ABB RAPID module: PRG_MVT.mod

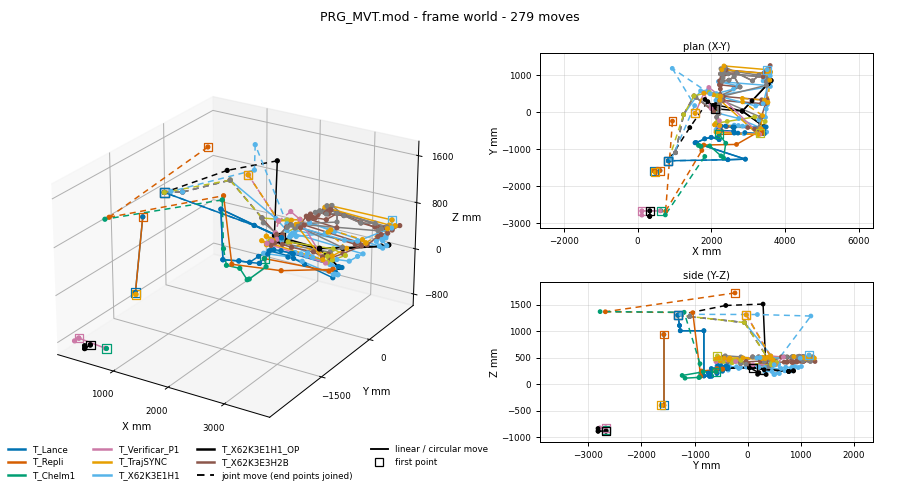
[picture p0: tool path of PRG_MVT.mod in frame world, 279 of 334 moves have a stored position in this frame; points joined in program order, loops and branches not executed]
%%%
  VERSION:1
  LANGUAGE:ENGLISH
%%%

MODULE PRG_MVT
  !********************************************
  !*                                          *
  !*      ABB--PROMIA--50.xx                  *
  !*                                          *
  !* Module Programme de mouvement            *
  !* Baie de commande de type IRC5            *
  !* Mono-robot                               *
  !********************************************
  !
  !=========================
  ! Donnees de type tooldata
  !=========================
  ! Outil par défaut pour T_Repli, T_Lance et trajs de Maintenance
  ! Les données de charge sont à renseigner !
  TASK PERS tooldata Tool_defaut:=[TRUE,[[0,0,0],[1,0,0,0]],[274,[0,0,0.001],[1,0,0,0],24.55,73.06,97.5]];
  ! Les données de charge et référentiels sont à renseigner !
  TASK PERS tooldata Tool_Pince1:=[TRUE,[[-1102.56,2.69854,432.58],[0.000350004,0,1,0]],[274,[0,0,0.001],[1,0,0,0],24.55,73.06,97.5]];
  TASK PERS tooldata Tool_Pince2:=[TRUE,[[0,0,0],[1,0,0,0]],[0.001,[0,0,0.001],[1,0,0,0],0,0,0]];
  TASK PERS tooldata Tool_Pince3:=[TRUE,[[0,0,0],[1,0,0,0]],[0.001,[0,0,0.001],[1,0,0,0],0,0,0]];
  TASK PERS tooldata Tool_Pince4:=[TRUE,[[0,0,0],[1,0,0,0]],[0.001,[0,0,0.001],[1,0,0,0],0,0,0]];
	TASK PERS tooldata Tool_etalonR1:=[TRUE,[[0,0,0],[1,0,0,0]],[0.001,[0,0,0.001],[1,0,0,0],0,0,0]];
  TASK PERS tooldata Tool_R1:=[TRUE,[[0,0,0],[1,0,0,0]],[0.001,[0,0,0.001],[1,0,0,0],0,0,0]];
  TASK PERS tooldata tMaxMotion:=[TRUE,[[-1102.56,2.69854,432.58],[0.000350004,0,1,0]],[0.001,[0,0,0.001],[1,0,0,0],0,0,0]];
  TASK PERS tooldata toolAtual:=[TRUE,[[0,0,0],[1,0,0,0]],[274,[0,0,0.001],[1,0,0,0],24.55,73.06,97.5]];
  PERS tooldata Temp_tool:=[TRUE,[[0,0,0],[1,0,0,0]],[0.001,[0,0,0.001],[1,0,0,0],0,0,0]];
  TASK PERS tooldata Pince1:=[TRUE,[[-1100.74,0,428.94],[0,0,1,0]],[274,[0,0,0.001],[1,0,0,0],24.55,73.06,97.5]];
  !
  !=========================
  ! Donnees de type wobjdata
  !=========================
  PERS wobjdata wobj_X62:=[FALSE,TRUE,"",[[0,0,0],[1,0,0,0]],[[2652.5,-1847.7,-1638.89],[0.737289,0.000738386,0.00238165,0.675573]]];
  TASK PERS wobjdata w_A11:=[FALSE,TRUE,"",[[723.52,3.59082,586.622],[0.104509,0.031933,0.994006,-0.00335437]],[[0,0,0],[0,1,0,0]]];
  TASK PERS wobjdata W_A21:=[FALSE,TRUE,"",[[723.52,3.59,586.62],[1,0,0,0]],[[0,0,0],[0,1,0,0]]];
  PERS wobjdata Temp_wobj:=[FALSE,TRUE,"",[[0,0,0],[1,0,0,0]],[[0,0,0],[1,0,0,0]]];
  PERS wobjdata Temp2_wobj:=[FALSE,TRUE,"",[[0,0,0],[1,0,0,0]],[[0,0,0],[1,0,0,0]]];
  TASK PERS wobjdata wobjAtual:=[FALSE,TRUE,"",[[0,0,0],[1,0,0,0]],[[0,0,0],[1,0,0,0]]];
  PERS wobjdata wobj_XDF:=[False,True,"",[[2664.9690,-1849.2940,-1633.2210],[0.737546,-0.004241,-0.002957,0.675277]],[[0,0,0],[1,0,0,0]]];
  !
  !=========================
  ! Donnees de type robtarget
  !=========================
  CONST robtarget pInicioX62_Pinca1:=[[366.51,1868.19,2935],[0.00946049,0.00387218,0.00595509,0.99993],[-1,-1,0,0],[29.4996,9E+09,9E+09,9E+09,9E+09,9E+09]];
  CONST robtarget pReferenciaPinca1:=[[117.16,-2786.22,-820.12],[0.578822,-0.00575624,0.000186763,-0.815434],[-1,-1,0,0],[72.8969,9E+09,9E+09,9E+09,9E+09,9E+09]];
  CONST robtarget pFresaPinca1:=[[330.76,-2818.92,-832.36],[0.67068,-0.00156521,-0.011854,-0.741651],[-1,0,0,0],[22.3121,9E+09,9E+09,9E+09,9E+09,9E+09]];
  CONST robtarget pTrocaEletrodosPinca1:=[[634.22,-2665.42,-865.34],[0.767575,-0.0054113,0.00150274,-0.640935],[-1,-1,0,0],[129.398,9E+09,9E+09,9E+09,9E+09,9E+09]];
  !

  !
  !=========================
  ! Donnees de type robtarget
  !=========================
  !Option Securité
  CONST jointtarget pPSync:=[[-74.4391,71.8518,8.78224,-3.78008,9.21547,38.5548],[72.8966,9E+09,9E+09,9E+09,9E+09,9E+09]];
  !
  !=========================
  ! Donnees de type bool
  !=========================
  PERS bool EPSRequest:=FALSE;
  !
  !-----------------------
  !     T_X62K3E1H1
  !-----------------------
  CONST robtarget lscs1002841400:=[[1321.80,-611.52,1989.42],[0.57763,-0.0127115,0.00458018,-0.816187],[-1,-1,0,0],[34.9983,9E+09,9E+09,9E+09,9E+09,9E+09]];
  CONST robtarget lscs1002841500:=[[1421.03,-636.06,1985.03],[0.577855,-0.0132046,0.00335794,-0.816026],[-1,-1,0,0],[34.9978,9E+09,9E+09,9E+09,9E+09,9E+09]];
  CONST robtarget lscs1002841900:=[[2124.39,-642.18,1983.84],[0.696596,0.0227135,0.0233793,-0.716723],[0,0,0,0],[34.9999,9E+09,9E+09,9E+09,9E+09,9E+09]];
  CONST robtarget lscs1002842000:=[[2228.68,-635.15,1986.45],[0.695583,0.0213858,0.0221666,-0.717786],[0,0,0,0],[35.0049,9E+09,9E+09,9E+09,9E+09,9E+09]];
  CONST robtarget lscs1002842300:=[[2641.55,-631.88,1984.23],[0.78191,0.0244769,0.0194947,-0.622606],[0,0,0,0],[20,9E+09,9E+09,9E+09,9E+09,9E+09]];
  CONST robtarget lscs1002842400:=[[2740.12,-630.61,1983.50],[0.787083,0.0248153,0.0202104,-0.616017],[0,0,0,0],[34.9988,9E+09,9E+09,9E+09,9E+09,9E+09]];
  CONST robtarget lscs1003265500:=[[1660.38,-715.96,1974.39],[0.623818,6.28508E-06,9.80078E-06,-0.781569],[0,-1,0,0],[35,9E+09,9E+09,9E+09,9E+09,9E+09]];
  CONST robtarget lscs1003265600:=[[1771.68,-715.35,1974.08],[0.641583,2.04864E-06,1.74234E-06,-0.767054],[0,-1,0,0],[35,9E+09,9E+09,9E+09,9E+09,9E+09]];
  CONST robtarget lscs1003265800:=[[2000.05,-716.75,1973.15],[0.67611,2.28831E-06,2.51046E-06,-0.736801],[0,-1,0,0],[34.9998,9E+09,9E+09,9E+09,9E+09,9E+09]];
  CONST robtarget lscs1003265900:=[[2103.17,-716.71,1973.07],[0.692842,6.80056E-06,1.10347E-05,-0.72109],[0,-1,0,0],[34.9998,9E+09,9E+09,9E+09,9E+09,9E+09]];
  CONST robtarget lscs1003266000:=[[2247.94,-712.34,1973.89],[0.709194,1.03549E-05,1.67342E-05,-0.705013],[0,-1,0,0],[34.9997,9E+09,9E+09,9E+09,9E+09,9E+09]];
  CONST robtarget lscs1003266100:=[[2332.06,-711.17,1972.75],[0.725199,1.11717E-05,1.69368E-05,-0.688539],[0,-1,0,0],[35,9E+09,9E+09,9E+09,9E+09,9E+09]];
  CONST robtarget lscs1003266200:=[[2415.91,-712.40,1971.62],[0.740802,6.31206E-07,-8.02992E-07,-0.671724],[0,-1,0,0],[35.0003,9E+09,9E+09,9E+09,9E+09,9E+09]];
  CONST robtarget lscs1003267400:=[[2515.38,-713.65,1970.65],[0.75603,-5.40779E-06,-9.51741E-06,-0.654537],[0,-1,0,0],[35,9E+09,9E+09,9E+09,9E+09,9E+09]];
  CONST robtarget lscs1003267500:=[[2614.89,-713.96,1971.44],[0.770849,8.75642E-06,1.09504E-05,-0.637018],[0,-1,0,0],[34.9997,9E+09,9E+09,9E+09,9E+09,9E+09]];
  CONST robtarget lscs1003267600:=[[2753.83,-713.47,1973.81],[0.787351,1.19686E-07,-7.7226E-06,-0.616505],[0,-1,0,0],[34.9996,9E+09,9E+09,9E+09,9E+09,9E+09]];
  CONST robtarget lscs1003267700:=[[2860.11,-710.59,1972.43],[0.787349,7.34808E-06,1.07537E-05,-0.616508],[0,-1,0,0],[35.0003,9E+09,9E+09,9E+09,9E+09,9E+09]];
  CONST robtarget lscs1003268200:=[[2954.09,-709.12,1972.24],[0.797982,-2.34679E-06,-6.61137E-06,-0.602681],[0,-1,0,0],[34.9997,9E+09,9E+09,9E+09,9E+09,9E+09]];
  CONST robtarget lscs1004621400:=[[1320.78,-635.11,1988.81],[0.577563,-0.00428276,0.010528,-0.816267],[-1,-1,0,0],[34.9983,9E+09,9E+09,9E+09,9E+09,9E+09]];
  CONST robtarget lscs1005331700:=[[1371.89,-717.33,1972.12],[0.595248,1.0937E-05,1.49243E-05,-0.803542],[-1,-1,0,0],[35.0037,9E+09,9E+09,9E+09,9E+09,9E+09]];
  CONST robtarget lscs2002842100:=[[2131.94,651.05,1966.73],[0.600981,-0.019579,-0.0260102,-0.7986],[0,-1,0,0],[25.7552,9E+09,9E+09,9E+09,9E+09,9E+09]];
  CONST robtarget lscs2002842200:=[[2234.34,649.61,1967.17],[0.613888,-0.0189544,-0.024229,-0.788794],[0,-1,0,0],[35.0005,9E+09,9E+09,9E+09,9E+09,9E+09]];
  CONST robtarget lscs2002842500:=[[2637.04,646.84,1973.10],[0.920442,-0.0269256,-0.00783123,-0.389872],[0,-1,-1,0],[33.1616,9E+09,9E+09,9E+09,9E+09,9E+09]];
  CONST robtarget lscs2003266400:=[[1657.98,727.29,1955.98],[0.356059,6.94468E-07,9.41827E-06,-0.934464],[0,0,0,0],[34.9945,9E+09,9E+09,9E+09,9E+09,9E+09]];
  CONST robtarget lscs2003266500:=[[1770.24,729.39,1956.83],[0.388522,1.29051E-06,-2.04438E-06,-0.92144],[0,0,0,0],[34.9997,9E+09,9E+09,9E+09,9E+09,9E+09]];
  CONST robtarget lscs2003266700:=[[1997.48,731.61,1956.90],[0.4602,4.00795E-06,-1.13671E-05,-0.887816],[0,0,0,0],[35.0891,9E+09,9E+09,9E+09,9E+09,9E+09]];
  CONST robtarget lscs2003266800:=[[2112.90,726.36,1955.43],[0.601155,1.22632E-06,9.81834E-06,-0.799133],[0,0,0,0],[35.0002,9E+09,9E+09,9E+09,9E+09,9E+09]];
  CONST robtarget lscs2003266900:=[[2249.72,730.07,1955.35],[0.614381,1.7781E-06,2.41043E-05,-0.789009],[0,0,0,0],[34.9999,9E+09,9E+09,9E+09,9E+09,9E+09]];
  CONST robtarget lscs2003267000:=[[2334.19,729.87,1957.44],[0.614386,-1.46543E-06,1.51219E-06,-0.789006],[0,0,0,0],[35.002,9E+09,9E+09,9E+09,9E+09,9E+09]];
  CONST robtarget lscs2003267100:=[[2418.69,727.31,1957.28],[0.670217,2.34267E-06,1.10938E-05,-0.742166],[0,0,0,0],[35,9E+09,9E+09,9E+09,9E+09,9E+09]];
  CONST robtarget lscs2003267800:=[[2517.33,728.02,1957.52],[0.712352,3.39692E-06,1.72802E-05,-0.701822],[0,0,0,0],[35,9E+09,9E+09,9E+09,9E+09,9E+09]];
  CONST robtarget lscs2003267900:=[[2618.90,732.56,1958.73],[0.92597,1.3493E-05,8.03361E-06,-0.377598],[0,-1,-1,0],[50.0003,9E+09,9E+09,9E+09,9E+09,9E+09]];
  CONST robtarget lscsd004573702:=[[1500.55,728.22,1952.50],[0.327808,2.82413E-06,-3.88473E-07,-0.944744],[0,0,0,0],[35.0009,9E+09,9E+09,9E+09,9E+09,9E+09]];
  CONST robtarget lscsg004573701:=[[1490.46,-715.35,1972.01],[0.605617,0.0139801,0.0105122,-0.795564],[-1,0,0,0],[34.9991,9E+09,9E+09,9E+09,9E+09,9E+09]];
  CONST robtarget lspac002878500:=[[1419.00,-536.94,1995.23],[0.572412,-0.0117175,0.00271518,-0.819878],[0,-1,0,0],[24.6351,9E+09,9E+09,9E+09,9E+09,9E+09]];
  CONST robtarget lspac002878600:=[[1417.58,-399.17,2001.89],[0.554961,-0.011186,0.00127143,-0.8318],[0,-1,0,0],[27.0922,9E+09,9E+09,9E+09,9E+09,9E+09]];
  CONST robtarget lspac002878700:=[[1416.53,-283.20,2005.54],[0.539023,-0.00172498,0.00603882,-0.842268],[0,-1,0,0],[22.9219,9E+09,9E+09,9E+09,9E+09,9E+09]];
  CONST robtarget lspac002878800:=[[1416.52,-204.20,2006.05],[0.527512,-0.00580073,0.00167739,-0.849526],[0,-1,0,0],[20.8186,9E+09,9E+09,9E+09,9E+09,9E+09]];

  CONST robtarget lspac002878900:=[[1416.87,-59.54,2005.71],[0.445099,0.000472,0.001718,-0.89548],[0,0,0,0],[35.002,9E+09,9E+09,9E+09,9E+09,9E+09]];
  CONST robtarget lspac002879000:=[[1416.21,53.99,2003.54],[0.445095,-0.001082,-0.001403,-0.895482],[0,-1,0,0],[27.999,9E+09,9E+09,9E+09,9E+09,9E+09]];
  CONST robtarget lspac002879100:=[[1417.29,167.25,2000.96],[0.418464,-0.003529,-0.007686,-0.908194],[0,-1,0,0],[35,9E+09,9E+09,9E+09,9E+09,9E+09]];
  CONST robtarget lspac002879200:=[[1416.66,280.75,1998.11],[0.370926,-0.005338,-0.013272,-0.928552],[0,-1,0,0],[35,9E+09,9E+09,9E+09,9E+09,9E+09]];
  CONST robtarget lspac002879300:=[[1416.64,393.28,1993.21],[0.370888,-0.007028,-0.017515,-0.928486],[0,-1,0,0],[35.004,9E+09,9E+09,9E+09,9E+09,9E+09]];
  CONST robtarget lspac002879400:=[[1417.48,505.46,1988.3],[0.371815,-0.009151,-0.022849,-0.927981],[0,-1,0,0],[35.002,9E+09,9E+09,9E+09,9E+09,9E+09]];
  CONST robtarget lscs2002841700:=[[1425.2,650.88,1974.99],[0.292836,-0.009125,-0.029745,-0.955656],[0,-1,0,0],[35,9E+09,9E+09,9E+09,9E+09,9E+09]];
  CONST robtarget lscs2004621500:=[[1322.81,651.07,1978.03],[0.285706,-0.009516,-0.031739,-0.957744],[0,-1,0,0],[37.176,9E+09,9E+09,9E+09,9E+09,9E+09]];
  CONST robtarget lscs2002841600:=[[1322.39,627.55,1981.36],[0.302378,-0.010051,-0.031649,-0.95261],[0,-1,0,0],[35,9E+09,9E+09,9E+09,9E+09,9E+09]];
  CONST robtarget lspac002883300:=[[1326.62,507.5,1989.98],[0.308491,-0.007592,-0.023435,-0.950908],[0,-1,0,0],[23.854,9E+09,9E+09,9E+09,9E+09,9E+09]];
  CONST robtarget lspac002883200:=[[1325.86,394.19,1995.58],[0.331525,-0.006266,-0.017813,-0.943257],[0,-1,0,0],[23.958,9E+09,9E+09,9E+09,9E+09,9E+09]];

  CONST robtarget lspac002883100:=[[1325.42,281.32,1997.89],[0.419379,-0.005519,-0.011953,-0.907716],[0,-1,0,0],[25.495,25.495,9E+09,9E+09,9E+09,9E+09]];
  CONST robtarget lspac002882400:=[[1321.76,-509.09,1996.03],[0.531284,-0.00843427,0.00739349,-0.84712],[0,-1,0,0],[35.0007,9E+09,9E+09,9E+09,9E+09,9E+09]];
  CONST robtarget lspac002882500:=[[1324.54,-396.08,2000.52],[0.51375,-0.00327198,-0.0104843,-0.85787],[0,0,0,0],[34.9986,9E+09,9E+09,9E+09,9E+09,9E+09]];
  CONST robtarget lspac002882600:=[[1324.67,-284.50,2002.23],[0.496324,0.000459301,-0.00172718,-0.868135],[0,0,0,0],[34.9989,9E+09,9E+09,9E+09,9E+09,9E+09]];
  CONST robtarget lspac002882700:=[[1324.62,-171.83,2005.66],[0.478463,-0.00395536,-0.0119621,-0.878018],[0,-1,0,0],[24.4112,9E+09,9E+09,9E+09,9E+09,9E+09]];
  CONST robtarget lspac002882800:=[[1324.87,-57.50,2005.46],[0.460554,-0.0108643,-0.00417129,-0.887556],[0,-1,0,0],[35.0038,9E+09,9E+09,9E+09,9E+09,9E+09]];
  CONST robtarget lspac002882900:=[[1324.13,55.63,2003.75],[0.44275,-0.00105814,-0.00139436,-0.896644],[0,-1,0,0],[20.988,9E+09,9E+09,9E+09,9E+09,9E+09]];
  CONST robtarget lspac002883000:=[[1324.03,167.68,2002.17],[0.419385,-0.00274683,-0.00713244,-0.907777],[0,-1,0,0],[19.1411,9E+09,9E+09,9E+09,9E+09,9E+09]];
  CONST robtarget lspac002900900:=[[2226.97,-511.07,1992.43],[0.695722,0.0173592,0.0179165,-0.717878],[0,0,0,0],[35.0017,9E+09,9E+09,9E+09,9E+09,9E+09]];
  CONST robtarget lspac002901000:=[[2226.48,-365.82,1995.55],[0.696043,0.0128999,0.0133004,-0.717761],[0,0,0,0],[34.9992,9E+09,9E+09,9E+09,9E+09,9E+09]];
  CONST robtarget lspac002901100:=[[2225.60,-228.43,1999.39],[0.69581,0.00731454,0.00755639,-0.718149],[0,0,0,0],[35.0004,9E+09,9E+09,9E+09,9E+09,9E+09]];
  CONST robtarget lspac002901300:=[[2225.20,24.47,1997.06],[0.695924,-0.00113677,-0.00115838,-0.718113],[0,-1,0,0],[35.0004,9E+09,9E+09,9E+09,9E+09,9E+09]];
  CONST robtarget lspac002901600:=[[2225.18,226.53,1992.98],[0.695884,-0.00731719,-0.00753954,-0.718077],[0,-1,0,0],[35.0003,9E+09,9E+09,9E+09,9E+09,9E+09]];
  CONST robtarget lspac002901700:=[[2227.57,364.45,1984.47],[0.695822,-0.0128824,-0.0132698,-0.717977],[0,-1,0,0],[35.0013,9E+09,9E+09,9E+09,9E+09,9E+09]];
  CONST robtarget lspac002901800:=[[2227.15,509.55,1976.50],[0.614039,-0.0153147,-0.0196554,-0.788882],[0,-1,0,0],[34.9978,9E+09,9E+09,9E+09,9E+09,9E+09]];
  CONST robtarget lspac002904100:=[[2126.95,-510.92,1993.00],[0.702146,-0.00802476,-0.0133731,-0.711862],[0,-1,0,0],[34.998,9E+09,9E+09,9E+09,9E+09,9E+09]];
  CONST robtarget lspac002904200:=[[2129.65,-364.85,2000.21],[0.7056,-0.00721348,-0.00638237,-0.708545],[0,-1,0,0],[34.9979,9E+09,9E+09,9E+09,9E+09,9E+09]];
  CONST robtarget lspac002904300:=[[2129.80,-227.65,1999.07],[0.714409,0.00750987,0.00734911,-0.69965],[0,0,0,0],[22.0001,9E+09,9E+09,9E+09,9E+09,9E+09]];
  CONST robtarget lspac002904400:=[[2132.73,-25.26,1998.55],[0.682213,0.00111235,0.00119395,-0.731152],[0,0,0,0],[20.0001,9E+09,9E+09,9E+09,9E+09,9E+09]];
  CONST robtarget lspac002904600:=[[2133.65,228.53,1991.11],[0.682136,-0.00715952,-0.00768831,-0.73115],[0,-1,0,0],[23.0024,9E+09,9E+09,9E+09,9E+09,9E+09]];
  CONST robtarget lspac002904700:=[[2132.48,364.88,1986.15],[0.682017,-0.0126149,-0.0135198,-0.731103],[0,-1,0,0],[21.9995,9E+09,9E+09,9E+09,9E+09,9E+09]];
  CONST robtarget lspac002904800:=[[2133.45,510.43,1978.85],[0.681915,-0.0169944,-0.0182283,-0.731007],[0,-1,0,0],[20.5101,9E+09,9E+09,9E+09,9E+09,9E+09]];
  CONST robtarget lspac002905100:=[[2739.39,-510.19,1990.50],[0.787183,0.0196481,0.015397,-0.616215],[0,0,0,0],[34.9996,9E+09,9E+09,9E+09,9E+09,9E+09]];
  CONST robtarget lspac002906100:=[[2644.16,-510.46,1992.58],[0.793004,0.0197938,0.0151959,-0.608706],[0,0,0,0],[19.9993,9E+09,9E+09,9E+09,9E+09,9E+09]];
  CONST robtarget lspac002906200:=[[2643.42,-365.01,1995.40],[0.80405,0.0149065,0.0110176,-0.594273],[0,0,0,0],[30.3308,9E+09,9E+09,9E+09,9E+09,9E+09]];
  CONST robtarget lspac002906300:=[[2642.81,-227.08,2000.09],[0.814671,0.00856781,0.00608173,-0.579829],[0,0,-1,0],[38.4896,9E+09,9E+09,9E+09,9E+09,9E+09]];
  CONST robtarget lspac002906400:=[[2639.69,-24.86,1997.79],[0.835042,0.00138016,0.000921054,-0.550184],[0,-1,-1,0],[31.1701,9E+09,9E+09,9E+09,9E+09,9E+09]];
  CONST robtarget lspac002906600:=[[2642.07,228.52,1996.03],[0.854261,-0.00895447,-0.00544438,-0.51974],[0,-1,-1,0],[56.311,9E+09,9E+09,9E+09,9E+09,9E+09]];
  CONST robtarget lspac002906700:=[[2642.16,368.74,1991.45],[0.877971,-0.0162117,-0.00882183,-0.478359],[0,-1,-1,0],[25.0003,9E+09,9E+09,9E+09,9E+09,9E+09]];
  CONST robtarget lspac002906800:=[[2640.35,507.33,1982.42],[0.904527,-0.0225527,-0.010627,-0.425687],[0,-1,-1,0],[29.1146,9E+09,9E+09,9E+09,9E+09,9E+09]];
  CONST robtarget lspac006169900:=[[2225.43,89.14,1997.34],[0.695931,-0.00294883,-0.00302088,-0.718096],[0,-1,0,0],[35.0021,9E+09,9E+09,9E+09,9E+09,9E+09]];
  CONST robtarget lspac006170200:=[[2133.71,90.17,1997.24],[0.6822,-0.00290099,-0.00312195,-0.731154],[0,-1,0,0],[21.9945,9E+09,9E+09,9E+09,9E+09,9E+09]];
  CONST robtarget lspac006170400:=[[2641.02,91.45,1996.56],[0.844807,-0.0035688,-0.00227158,-0.535055],[0,-1,-1,0],[31.1277,9E+09,9E+09,9E+09,9E+09,9E+09]];
  CONST robtarget lspac006170500:=[[2226.35,-90.87,1999.36],[0.695897,0.00294943,0.00305218,-0.718129],[0,0,0,0],[34.9995,9E+09,9E+09,9E+09,9E+09,9E+09]];
  CONST robtarget lspac006170800:=[[2134.22,-89.69,2000.26],[0.720063,0.00306425,0.00294629,-0.693896],[0,0,0,0],[22,9E+09,9E+09,9E+09,9E+09,9E+09]];
  CONST robtarget lspac006171000:=[[2641.20,-82.11,1999.25],[0.824987,0.00352259,0.00243168,-0.565135],[0,0,-1,0],[38.713,9E+09,9E+09,9E+09,9E+09,9E+09]];
  !-----------------------
  !    T_X62K3E1H1_OP
  !-----------------------
  CONST robtarget lscs1003265700:=[[1886.36,-714.00,1973.66],[0.653882,-1.55351E-06,-1.78434E-06,-0.756597],[0,-1,0,0],[75.0001,9E+09,9E+09,9E+09,9E+09,9E+09]];
  CONST robtarget lscs2003266600:=[[1884.13,727.83,1956.34],[0.460207,5.49601E-07,1.78346E-06,-0.887812],[0,0,0,0],[74.9997,9E+09,9E+09,9E+09,9E+09,9E+09]];
  !-----------------------
  !    T_X62K3E23H2
  !-----------------------
  CONST robtarget lscs1002838100:=[[1326.03,-548.67,2179.62],[0.529877,0.0162447,0.0240929,-0.847577],[-1,0,0,0],[35.0008,9E+09,9E+09,9E+09,9E+09,9E+09]];
  CONST robtarget lscs1002838200:=[[1420.36,-572.64,2182.13],[0.520361,0.0154283,0.0248866,-0.853444],[0,0,0,0],[35.0001,9E+09,9E+09,9E+09,9E+09,9E+09]];
  CONST robtarget lscs1002838900:=[[2127.03,-573.84,2183.93],[0.703375,0.0176685,0.0238462,-0.710199],[0,0,0,0],[34.9991,9E+09,9E+09,9E+09,9E+09,9E+09]];
  CONST robtarget lscs1002839000:=[[2230.97,-578.10,2182.31],[0.695615,0.0204629,0.021045,-0.717815],[0,0,0,0],[46.4605,9E+09,9E+09,9E+09,9E+09,9E+09]];
  CONST robtarget lscs1002839300:=[[2853.37,-575.98,2185.81],[0.828085,0.0232734,0.0156745,-0.559901],[0,0,-1,0],[34.9997,9E+09,9E+09,9E+09,9E+09,9E+09]];
  CONST robtarget lscs1002839400:=[[2956.67,-579.33,2185.33],[0.856587,0.0240684,0.0144354,-0.515239],[0,0,-1,0],[40.0003,9E+09,9E+09,9E+09,9E+09,9E+09]];
  CONST robtarget lscs1002942300:=[[2626.98,-655.27,2171.32],[0.804153,-8.6074E-06,-1.1363E-05,-0.594422],[0,-1,-1,0],[34.9998,9E+09,9E+09,9E+09,9E+09,9E+09]];
  CONST robtarget lscs1002947100:=[[2738.19,-655.26,2169.96],[0.804153,4.11586E-06,4.76108E-06,-0.594422],[0,-1,0,0],[34.9992,9E+09,9E+09,9E+09,9E+09,9E+09]];
  CONST robtarget lscs1002947200:=[[2809.98,-656.04,2169.47],[0.81522,4.45343E-06,6.51458E-06,-0.579152],[0,-1,-1,0],[39.9989,9E+09,9E+09,9E+09,9E+09,9E+09]];
  CONST robtarget lscs1002947300:=[[2974.64,-656.15,2165.68],[0.825996,0.00211954,0.00310276,-0.563664],[0,-1,0,0],[35.0001,9E+09,9E+09,9E+09,9E+09,9E+09]];
  CONST robtarget lscs1002947400:=[[3079.28,-658.62,2169.89],[0.823766,3.1187E-06,2.90278E-06,-0.56693],[0,-1,0,0],[35.0004,9E+09,9E+09,9E+09,9E+09,9E+09]];
  CONST robtarget lscs2002838300:=[[1325.75,565.96,2167.59],[0.309017,-0.00800614,-0.0278437,-0.950615],[0,-1,0,0],[34.9998,9E+09,9E+09,9E+09,9E+09,9E+09]];
  CONST robtarget lscs2002838400:=[[1427.30,583.02,2168.42],[0.340966,-0.00978532,-0.0275895,-0.93962],[0,-1,0,0],[35.0004,9E+09,9E+09,9E+09,9E+09,9E+09]];
  CONST robtarget lscs2002839100:=[[2133.43,593.10,2171.39],[0.601042,-0.0175714,-0.0234515,-0.79868],[0,-1,0,0],[34.9998,9E+09,9E+09,9E+09,9E+09,9E+09]];
  CONST robtarget lscs2002839200:=[[2231.78,587.70,2169.83],[0.613987,-0.017952,-0.0231091,-0.788773],[0,-1,0,0],[35.002,9E+09,9E+09,9E+09,9E+09,9E+09]];
  CONST robtarget lscs2002839500:=[[2855.38,589.72,2170.01],[0.936255,-0.0262308,-0.0098444,-0.350202],[0,-1,-1,0],[34.9994,9E+09,9E+09,9E+09,9E+09,9E+09]];
  CONST robtarget lscs2002839600:=[[2955.83,589.35,2166.58],[0.92948,-0.0260606,-0.0103697,-0.367804],[0,-1,-1,0],[34.9989,9E+09,9E+09,9E+09,9E+09,9E+09]];
  CONST robtarget lscs2002942400:=[[1656.42,669.92,2155.44],[0.381231,-0.00569286,-0.00235086,-0.924459],[0,-1,0,0],[34.9996,9E+09,9E+09,9E+09,9E+09,9E+09]];
  CONST robtarget lscs2002947700:=[[2974.90,666.23,2157.26],[0.956656,1.24176E-06,-1.32246E-06,-0.291221],[0,-1,-1,0],[35.0004,9E+09,9E+09,9E+09,9E+09,9E+09]];
  CONST robtarget lscs2002948300:=[[2748.62,669.50,2157.71],[0.934712,-0.0166626,-0.00769493,-0.354931],[0,-1,-1,0],[35.0013,9E+09,9E+09,9E+09,9E+09,9E+09]];
  CONST robtarget lscs2002948400:=[[2839.99,664.03,2158.93],[0.930824,-0.0127707,-0.0125728,-0.365028],[0,0,-1,0],[35.0004,9E+09,9E+09,9E+09,9E+09,9E+09]];
  CONST robtarget lscsd002940401:=[[1769.97,-653.94,2173.43],[0.620932,0.00566687,0.00449122,-0.783831],[0,0,0,0],[34.9999,9E+09,9E+09,9E+09,9E+09,9E+09]];
  CONST robtarget lscsd002940501:=[[1884.80,-654.85,2173.58],[0.644987,0.00505808,0.00427322,-0.764165],[0,0,0,0],[35.0001,9E+09,9E+09,9E+09,9E+09,9E+09]];
  CONST robtarget lscsd002940601:=[[1997.83,-655.31,2171.98],[0.668329,0.0125735,0.0113003,-0.743674],[0,0,0,0],[34.9999,9E+09,9E+09,9E+09,9E+09,9E+09]];
  CONST robtarget lscsd002940701:=[[2072.98,-654.70,2171.88],[0.693589,0.00912135,0.00877874,-0.72026],[0,0,0,0],[34.9996,9E+09,9E+09,9E+09,9E+09,9E+09]];
  CONST robtarget lscsd002940801:=[[2291.22,-655.36,2173.59],[0.713321,-2.28443E-06,-7.63419E-06,-0.700837],[0,-1,0,0],[42.9768,9E+09,9E+09,9E+09,9E+09,9E+09]];
  CONST robtarget lscsd002940901:=[[2332.00,-657.77,2175.31],[0.732657,-1.18719E-05,-1.97091E-05,-0.680598],[0,-1,0,0],[34.9966,9E+09,9E+09,9E+09,9E+09,9E+09]];
  CONST robtarget lscsd002941001:=[[2417.36,-655.05,2172.07],[0.751432,-1.33253E-05,-2.16398E-05,-0.659811],[0,-1,0,0],[34.9999,9E+09,9E+09,9E+09,9E+09,9E+09]];
  CONST robtarget lscsd002941201:=[[2527.31,-655.34,2171.69],[0.769614,-1.00867E-05,-1.72388E-05,-0.638509],[0,-1,0,0],[34.9996,9E+09,9E+09,9E+09,9E+09,9E+09]];
  CONST robtarget lscsg002940402:=[[1769.70,672.77,2160.05],[0.460134,-0.0158576,-0.00820563,-0.88767],[0,-1,0,0],[35.0002,9E+09,9E+09,9E+09,9E+09,9E+09]];
  CONST robtarget lscsg002940502:=[[1885.15,669.83,2160.62],[0.460128,-0.0169626,-0.00877886,-0.887647],[0,-1,0,0],[35.0014,9E+09,9E+09,9E+09,9E+09,9E+09]];
  CONST robtarget lscsg002940602:=[[1997.71,669.05,2158.61],[0.460152,-0.0137371,-0.0071145,-0.887705],[0,-1,0,0],[35.0005,9E+09,9E+09,9E+09,9E+09,9E+09]];
  CONST robtarget lscsg002940702:=[[2082.50,666.45,2160.87],[0.602889,-0.0228712,-0.0226078,-0.797176],[0,-1,0,0],[35.0007,9E+09,9E+09,9E+09,9E+09,9E+09]];
  CONST robtarget lscsg002940802:=[[2252.27,665.75,2159.94],[0.61421,-0.0185701,-0.0144589,-0.788792],[0,-1,0,0],[35,9E+09,9E+09,9E+09,9E+09,9E+09]];
  CONST robtarget lscsg002940902:=[[2343.10,668.27,2161.44],[0.652027,-0.0113834,-0.009793,-0.758047],[0,-1,0,0],[34.9994,9E+09,9E+09,9E+09,9E+09,9E+09]];
  CONST robtarget lscsg002941002:=[[2427.58,668.43,2156.81],[0.651992,-0.0136378,-0.00997592,-0.758038],[0,-1,0,0],[34.9996,9E+09,9E+09,9E+09,9E+09,9E+09]];
  CONST robtarget lscsg002941202:=[[2540.60,667.51,2158.29],[0.712276,-0.0103406,-0.0104855,-0.701745],[0,-1,0,0],[34.9995,9E+09,9E+09,9E+09,9E+09,9E+09]];
  CONST robtarget lscsg002941302:=[[2642.64,666.07,2158.11],[0.921929,-0.0056908,-0.0130385,-0.387097],[0,0,-1,0],[40.0002,9E+09,9E+09,9E+09,9E+09,9E+09]];
  CONST robtarget lscsg002952001:=[[3180.19,-652.97,2171.39],[0.833497,0.00504659,0.00761065,-0.552449],[0,0,0,0],[39.9991,9E+09,9E+09,9E+09,9E+09,9E+09]];
  CONST robtarget lspac002867100:=[[1417.73,-475.90,2184.09],[0.520497,0.0116919,0.0184006,-0.853585],[0,0,0,0],[35.0004,9E+09,9E+09,9E+09,9E+09,9E+09]];
  CONST robtarget lspac002867200:=[[1417.86,-380.26,2188.10],[0.520507,0.0116874,0.0183921,-0.85358],[0,0,0,0],[34.9993,9E+09,9E+09,9E+09,9E+09,9E+09]];
  CONST robtarget lspac002867300:=[[1418.70,-201.15,2191.52],[0.488303,0.00480831,0.00861262,-0.872618],[0,0,0,0],[35.0007,9E+09,9E+09,9E+09,9E+09,9E+09]];
  CONST robtarget lspac002867400:=[[1421.87,89.01,2189.93],[0.460915,-0.00119251,-0.00230585,-0.887441],[0,-1,0,0],[34.9984,9E+09,9E+09,9E+09,9E+09,9E+09]];
  CONST robtarget lspac002867500:=[[1424.88,192.62,2187.87],[0.460879,-0.00466,-0.00864293,-0.887409],[0,-1,0,0],[34.9982,9E+09,9E+09,9E+09,9E+09,9E+09]];
  CONST robtarget lspac002867600:=[[1424.55,389.96,2176.75],[0.399559,-0.00737384,-0.0168728,-0.916523],[0,-1,0,0],[34.997,9E+09,9E+09,9E+09,9E+09,9E+09]];
  CONST robtarget lspac002867700:=[[1425.34,474.84,2177.44],[0.353858,-0.00732357,-0.0204989,-0.935046],[0,-1,0,0],[34.9995,9E+09,9E+09,9E+09,9E+09,9E+09]];
  CONST robtarget lspac002870900:=[[1319.75,-557.12,2179.67],[0.529934,0.0144646,0.0217019,-0.847638],[-1,0,0,0],[36.3642,9E+09,9E+09,9E+09,9E+09,9E+09]];
  CONST robtarget lspac002871000:=[[1322.01,-452.05,2186.77],[0.520789,-0.00501219,0.00852188,-0.853628],[0,-1,0,0],[34.9994,9E+09,9E+09,9E+09,9E+09,9E+09]];
  CONST robtarget lspac002871100:=[[1322.04,-350.17,2188.84],[0.520733,-0.00261869,0.00698991,-0.853687],[0,-1,0,0],[34.9997,9E+09,9E+09,9E+09,9E+09,9E+09]];
  CONST robtarget lspac002871200:=[[1323.00,-251.05,2188.86],[0.488365,-0.00336017,0.00559701,-0.872615],[0,-1,0,0],[34.9994,9E+09,9E+09,9E+09,9E+09,9E+09]];
  CONST robtarget lspac002871300:=[[1323.51,-152.97,2191.83],[0.488352,-0.00560002,0.000560971,-0.872629],[0,-1,0,0],[35.0008,9E+09,9E+09,9E+09,9E+09,9E+09]];
  CONST robtarget lspac002871400:=[[1321.82,-54.05,2191.69],[0.460818,-0.0131272,-0.00586989,-0.887378],[0,-1,0,0],[34.9994,9E+09,9E+09,9E+09,9E+09,9E+09]];
  CONST robtarget lspac002871500:=[[1322.40,52.44,2189.02],[0.460864,-0.0101083,-0.00615694,-0.887392],[0,-1,0,0],[34.9997,9E+09,9E+09,9E+09,9E+09,9E+09]];
  CONST robtarget lspac002871600:=[[1324.07,151.29,2186.20],[0.418098,-0.0112449,-0.0109454,-0.908267],[0,-1,0,0],[35.0002,9E+09,9E+09,9E+09,9E+09,9E+09]];
  CONST robtarget lspac002871700:=[[1323.04,250.15,2182.92],[0.402189,-0.0125378,-0.0154928,-0.91534],[0,-1,0,0],[34.9986,9E+09,9E+09,9E+09,9E+09,9E+09]];
  CONST robtarget lspac002871800:=[[1323.80,348.44,2179.41],[0.40225,-0.010811,-0.0165279,-0.915317],[0,-1,0,0],[34.998,9E+09,9E+09,9E+09,9E+09,9E+09]];
  CONST robtarget lspac002871900:=[[1324.63,467.15,2175.31],[0.357237,-0.0131996,-0.0236411,-0.933622],[0,-1,0,0],[34.9997,9E+09,9E+09,9E+09,9E+09,9E+09]];
  CONST robtarget lspac002872000:=[[1325.26,522.33,2170.19],[0.312239,-0.0135515,-0.0251911,-0.949573],[0,-1,0,0],[34.9997,9E+09,9E+09,9E+09,9E+09,9E+09]];
  CONST robtarget lspac002889700:=[[2130.92,-449.96,2190.94],[0.708617,0.012701,0.0184545,-0.705237],[0,0,0,0],[34.9997,9E+09,9E+09,9E+09,9E+09,9E+09]];
  CONST robtarget lspac002889800:=[[2130.11,-305.14,2193.90],[0.713767,0.00843304,0.0142752,-0.700187],[0,-1,0,0],[34.9997,9E+09,9E+09,9E+09,9E+09,9E+09]];
  CONST robtarget lspac002889900:=[[2128.97,-200.46,2194.90],[0.718862,0.000396026,0.0121208,-0.695047],[0,-1,0,0],[34.9997,9E+09,9E+09,9E+09,9E+09,9E+09]];
  CONST robtarget lspac002890000:=[[2130.97,28.60,2195.63],[0.682194,-0.0055839,0.00217401,-0.731147],[0,-1,0,0],[35,9E+09,9E+09,9E+09,9E+09,9E+09]];
  CONST robtarget lspac002890100:=[[2132.58,200.68,2192.47],[0.682099,-0.009952,-0.0025133,-0.731188],[0,-1,0,0],[34.9997,9E+09,9E+09,9E+09,9E+09,9E+09]];
  CONST robtarget lspac002890200:=[[2132.13,305.50,2189.12],[0.681978,-0.0148022,-0.00770275,-0.731182],[0,-1,0,0],[35.0001,9E+09,9E+09,9E+09,9E+09,9E+09]];
  CONST robtarget lspac002890300:=[[2134.28,445.66,2181.49],[0.68176,-0.0222216,-0.00839884,-0.73119],[0,-1,0,0],[34.9995,9E+09,9E+09,9E+09,9E+09,9E+09]];
  CONST robtarget lspac002890400:=[[2225.77,-445.98,2189.55],[0.695756,0.0150473,0.0155268,-0.717953],[0,0,0,0],[35.002,9E+09,9E+09,9E+09,9E+09,9E+09]];
  CONST robtarget lspac002890500:=[[2224.97,-305.37,2193.33],[0.694114,0.00182386,0.00126215,-0.719862],[0,0,0,0],[35.0012,9E+09,9E+09,9E+09,9E+09,9E+09]];
  CONST robtarget lspac002890600:=[[2223.85,-200.64,2195.45],[0.695867,0.000467568,0.000933011,-0.71817],[0,-1,0,0],[34.9985,9E+09,9E+09,9E+09,9E+09,9E+09]];
  CONST robtarget lspac002890700:=[[2225.07,-15.49,2196.34],[0.695932,-0.00101749,-0.000863021,-0.718106],[0,-1,0,0],[34.9985,9E+09,9E+09,9E+09,9E+09,9E+09]];
  CONST robtarget lspac002890800:=[[2225.57,200.10,2191.69],[0.695909,-0.0076485,-0.00788185,-0.718046],[0,-1,0,0],[34.9988,9E+09,9E+09,9E+09,9E+09,9E+09]];
  CONST robtarget lspac002890900:=[[2226.51,306.30,2190.19],[0.695849,-0.0112182,-0.0115893,-0.718007],[0,-1,0,0],[35.0009,9E+09,9E+09,9E+09,9E+09,9E+09]];
  CONST robtarget lspac002891000:=[[2226.11,445.10,2179.90],[0.695774,-0.0150427,-0.0155104,-0.717936],[0,-1,0,0],[34.9999,9E+09,9E+09,9E+09,9E+09,9E+09]];
  CONST robtarget lspac002892500:=[[2855.43,-451.40,2191.40],[0.836183,0.0191768,0.0125763,-0.547971],[0,0,-1,0],[35,9E+09,9E+09,9E+09,9E+09,9E+09]];
  CONST robtarget lspac002892600:=[[2855.89,-305.04,2195.71],[0.843791,0.0129785,0.00818236,-0.536452],[0,0,-1,0],[35,9E+09,9E+09,9E+09,9E+09,9E+09]];
  CONST robtarget lspac002892700:=[[2856.68,-200.50,2197.82],[0.851203,0.00850307,0.0052359,-0.524742],[0,0,-1,0],[35,9E+09,9E+09,9E+09,9E+09,9E+09]];
  CONST robtarget lspac002892800:=[[2857.46,30.31,2195.22],[0.865427,-0.00929013,0.0027154,-0.500941],[0,-1,-1,0],[34.9999,9E+09,9E+09,9E+09,9E+09,9E+09]];
  CONST robtarget lspac002892900:=[[2858.72,196.22,2194.16],[0.878853,-0.0197125,0.00111028,-0.476683],[0,-1,-1,0],[34.9996,9E+09,9E+09,9E+09,9E+09,9E+09]];
  CONST robtarget lspac002893000:=[[2857.97,305.04,2188.48],[0.878566,-0.0134354,-0.00735434,-0.477376],[0,-1,-1,0],[35.001,9E+09,9E+09,9E+09,9E+09,9E+09]];
  CONST robtarget lspac002893100:=[[2856.71,445.31,2181.38],[0.918149,-0.0146585,0.00597393,-0.395919],[0,-1,-1,0],[35.0004,9E+09,9E+09,9E+09,9E+09,9E+09]];
  CONST robtarget lspac002893200:=[[2954.63,-444.86,2191.05],[0.852783,0.0177804,0.00907132,-0.521884],[0,0,-1,0],[35.0002,9E+09,9E+09,9E+09,9E+09,9E+09]];
  CONST robtarget lspac002893300:=[[2954.04,-305.19,2196.72],[0.856396,0.0131678,0.00787434,-0.516092],[0,0,-1,0],[35.0003,9E+09,9E+09,9E+09,9E+09,9E+09]];
  CONST robtarget lspac002893400:=[[2953.74,-202.66,2195.88],[0.872035,0.00874725,0.00491824,-0.489341],[0,0,-1,0],[34.9994,9E+09,9E+09,9E+09,9E+09,9E+09]];
  CONST robtarget lspac002893500:=[[2954.78,-16.65,2196.49],[0.881569,0.0199558,-0.00819289,-0.471562],[0,0,-1,0],[35.0002,9E+09,9E+09,9E+09,9E+09,9E+09]];
  CONST robtarget lspac002893600:=[[2953.28,200.20,2192.18],[0.891186,-0.00892448,-0.00454672,-0.453528],[0,-1,-1,0],[34.9998,9E+09,9E+09,9E+09,9E+09,9E+09]];
  CONST robtarget lspac002893700:=[[2954.54,304.77,2187.77],[0.895283,-0.0137113,-0.00687323,-0.445234],[0,-1,-1,0],[34.9998,9E+09,9E+09,9E+09,9E+09,9E+09]];
  CONST robtarget lspac002893800:=[[2954.09,442.89,2179.98],[0.903303,-0.0206959,-0.00979665,-0.428392],[0,-1,-1,0],[34.9998,9E+09,9E+09,9E+09,9E+09,9E+09]];
  CONST robtarget lspac004679300:=[[1419.40,-90.53,2191.96],[0.488332,0.00128769,0.00230418,-0.872654],[0,-1,0,0],[34.9956,9E+09,9E+09,9E+09,9E+09,9E+09]];
  CONST robtarget lspac006167600:=[[2224.59,89.55,2194.12],[0.695935,-0.00181934,-0.00185364,-0.7181],[0,-1,0,0],[35.0001,9E+09,9E+09,9E+09,9E+09,9E+09]];
  CONST robtarget lspac006167800:=[[2954.58,89.81,2198.74],[0.884135,-0.00232395,-0.00123696,-0.467224],[0,-1,-1,0],[34.9993,9E+09,9E+09,9E+09,9E+09,9E+09]];
  CONST robtarget lspac006168200:=[[2131.32,88.86,2194.81],[0.682203,-0.004364,0.000880584,-0.731149],[0,-1,0,0],[34.9991,9E+09,9E+09,9E+09,9E+09,9E+09]];
  CONST robtarget lspac006168400:=[[2857.92,89.99,2196.93],[0.872361,-0.00229199,-0.00127721,-0.488856],[0,-1,-1,0],[34.9996,9E+09,9E+09,9E+09,9E+09,9E+09]];
  CONST robtarget lspac006168800:=[[2225.08,-90.00,2196.69],[0.694408,0.00167789,-0.00658465,-0.71955],[0,0,0,0],[35.0001,9E+09,9E+09,9E+09,9E+09,9E+09]];
  CONST robtarget lspac006169000:=[[2954.99,-91.13,2196.49],[0.876984,0.00230734,0.00126586,-0.480513],[0,0,-1,0],[35.0002,9E+09,9E+09,9E+09,9E+09,9E+09]];
  CONST robtarget lspac006169400:=[[2130.79,-89.91,2196.61],[0.723873,-0.000942108,0.00452856,-0.689918],[0,-1,0,0],[35,9E+09,9E+09,9E+09,9E+09,9E+09]];
  CONST robtarget lspac006169600:=[[2858.97,-89.91,2198.38],[0.858431,0.0022495,0.00133534,-0.512922],[0,0,-1,0],[35.0014,9E+09,9E+09,9E+09,9E+09,9E+09]];
  CONST robtarget lspac006171300:=[[1419.08,-305.58,2188.48],[0.520609,0.00787595,0.0129187,-0.853661],[0,0,0,0],[35.0004,9E+09,9E+09,9E+09,9E+09,9E+09]];
  CONST robtarget lspac006171700:=[[1421.52,-2.47,2191.15],[0.460866,0.00121513,0.00235755,-0.887466],[0,0,0,0],[35.0001,9E+09,9E+09,9E+09,9E+09,9E+09]];
  CONST robtarget lspac006172100:=[[1424.14,305.04,2183.69],[0.445272,-0.00671443,-0.013478,-0.895269],[0,-1,0,0],[34.9998,9E+09,9E+09,9E+09,9E+09,9E+09]];
  !-----------------------
  !    T_X62K3E23H2_OP
  !-----------------------
  CONST robtarget lscs1004359200:=[[1491.83,-651.79,2172.44],[0.597781,-4.97762E-06,-7.37094E-06,-0.80166],[-1,-1,0,0],[39.9999,9E+09,9E+09,9E+09,9E+09,9E+09]];
  CONST robtarget lscs2004359300:=[[1497.46,666.14,2157.75],[0.339478,5.15567E-06,3.28474E-06,-0.940614],[0,0,0,0],[39.9999,9E+09,9E+09,9E+09,9E+09,9E+09]];
  CONST robtarget lscsd002940301:=[[1657.30,-654.86,2173.55],[0.605718,-9.11264E-06,-1.74615E-05,-0.79568],[0,-1,0,0],[40.0003,9E+09,9E+09,9E+09,9E+09,9E+09]];
  !-----------------------
  !    T_X62K3CC
  !-----------------------
  CONST robtarget lscs1002858200:=[[1321.92,-635.54,1985.86],[0.771868,0.0170389,0.0107964,-0.635462],[-1,-1,-1,0],[34.951,9E+09,9E+09,9E+09,9E+09,9E+09]];
  CONST robtarget lscs1004621800:=[[1320.01,-657.55,1986.16],[0.771868,0.0170267,0.0107917,-0.635463],[-1,-1,-1,0],[34.9538,9E+09,9E+09,9E+09,9E+09,9E+09]];
  CONST robtarget lscs2002858000:=[[1318.04,652.83,1975.04],[0.873219,-0.0172824,-0.01086,-0.486901],[-1,0,-1,0],[34.9997,9E+09,9E+09,9E+09,9E+09,9E+09]];
  CONST robtarget lscs2004621900:=[[1315.29,674.79,1973.05],[0.878232,-0.0119713,-0.0222557,-0.477568],[-1,0,-1,0],[34.9997,9E+09,9E+09,9E+09,9E+09,9E+09]];
  CONST robtarget lspac002883400:=[[1325.07,-510.35,1995.16],[0.781284,0.0207537,0.0165702,-0.623611],[-1,-1,-1,0],[35.0005,9E+09,9E+09,9E+09,9E+09,9E+09]];
  CONST robtarget lspac002883500:=[[1324.55,-397.08,1999.11],[0.808673,0.0158405,0.0115171,-0.587933],[-1,-1,-1,0],[35,9E+09,9E+09,9E+09,9E+09,9E+09]];
  CONST robtarget lspac002883600:=[[1323.60,-283.83,1998.42],[0.820293,0.0120305,0.00839675,-0.571755],[-1,-1,-1,0],[35,9E+09,9E+09,9E+09,9E+09,9E+09]];
  CONST robtarget lspac002883700:=[[1323.92,-170.33,1998.98],[0.824891,0.0066361,0.00455045,-0.565234],[-1,-1,-1,0],[35.0006,9E+09,9E+09,9E+09,9E+09,9E+09]];
  CONST robtarget lspac002883800:=[[1322.76,-57.01,1997.07],[0.823888,0.00270504,0.00186622,-0.566743],[-1,-1,-1,0],[34.9997,9E+09,9E+09,9E+09,9E+09,9E+09]];
  CONST robtarget lspac002883900:=[[1322.35,56.52,1994.83],[0.825628,-0.00266104,-0.00182578,-0.564206],[-1,-1,-1,0],[35.0008,9E+09,9E+09,9E+09,9E+09,9E+09]];
  CONST robtarget lspac002884000:=[[1322.07,169.79,1994.35],[0.833182,-0.000361833,0.00475025,-0.552979],[-1,-1,-1,0],[35.0003,9E+09,9E+09,9E+09,9E+09,9E+09]];
  CONST robtarget lspac002884100:=[[1320.96,283.89,1989.54],[0.869185,0.00505625,0.0293607,-0.493589],[-1,-1,-1,0],[34.9996,9E+09,9E+09,9E+09,9E+09,9E+09]];
  CONST robtarget lspac002884200:=[[1322.07,398.39,1986.31],[0.896394,0.0133055,0.0334012,-0.441798],[-1,-1,-1,0],[35.0003,9E+09,9E+09,9E+09,9E+09,9E+09]];
  CONST robtarget lspac002884300:=[[1321.53,510.04,1984.82],[0.863154,-0.00931482,-0.0136485,-0.50467],[-1,0,-1,0],[35.001,9E+09,9E+09,9E+09,9E+09,9E+09]];
  !-----------------------
  !    T_X62K3E3H2B
  !-----------------------
  CONST robtarget lscsg002940802_B:=[[2282.40,667.48,2160.68],[0.614127,-0.0211686,-0.0111228,-0.788845],[0,-1,0,0],[35.0005,9E+09,9E+09,9E+09,9E+09,9E+09]];
  CONST robtarget lscs1002839400_B:=[[2954.99,-548.18,2183.51],[0.856583,0.0240611,0.0144304,-0.515245],[0,0,-1,0],[35.0001,9E+09,9E+09,9E+09,9E+09,9E+09]];
  CONST robtarget lscs2002839600_B:=[[2955.01,564.28,2176.68],[0.920033,-0.0521134,-0.0265021,-0.387454],[0,-1,-1,0],[30,9E+09,9E+09,9E+09,9E+09,9E+09]];
  CONST robtarget lscs2002839500_B:=[[2854.51,566.35,2174.71],[0.930806,-0.0163607,-0.0434952,-0.362547],[0,0,-1,0],[35.0002,9E+09,9E+09,9E+09,9E+09,9E+09]];
  CONST robtarget lscs1002839300_B:=[[2857.59,-550.62,2182.29],[0.832504,0.028115,0.0314098,-0.552414],[0,0,-1,0],[30,9E+09,9E+09,9E+09,9E+09,9E+09]];
  CONST robtarget lscs1002839000_B:=[[2229.19,-547.05,2184.75],[0.695175,0.0321999,0.0324107,-0.717387],[0,0,0,0],[30,9E+09,9E+09,9E+09,9E+09,9E+09]];
  CONST robtarget lscs2002839200_B:=[[2232.29,564.59,2174.15],[0.695058,-0.0343763,-0.0362361,-0.717217],[0,-1,0,0],[30,9E+09,9E+09,9E+09,9E+09,9E+09]];
  CONST robtarget lscs2002839100_B:=[[2132.77,566.19,2177.4],[0.656827,-0.0453161,-0.046042,-0.751269],[0,-1,0,0],[30,9E+09,9E+09,9E+09,9E+09,9E+09]];
  CONST robtarget lscs1002838900_B:=[[2130.11,-546.81,2190.83],[0.708065,0.0276648,0.03349,-0.70481],[0,0,0,0],[30,9E+09,9E+09,9E+09,9E+09,9E+09]];
  CONST robtarget lscs1002838200_B:=[[1424.00,-548.33,2180.56],[0.519984,0.0269104,0.0318929,-0.853156],[0,0,0,0],[34.9992,9E+09,9E+09,9E+09,9E+09,9E+09]];
  CONST robtarget lspac006171300_B:=[[1423.18,-359.60,2188.77],[0.52057,0.00961868,0.0158056,-0.853619],[0,0,0,0],[34.9982,9E+09,9E+09,9E+09,9E+09,9E+09]];
  CONST robtarget lspac006172100_B:=[[1423.41,358.23,2182.53],[0.399539,-0.00737597,-0.0169085,-0.916531],[0,-1,0,0],[34.9998,9E+09,9E+09,9E+09,9E+09,9E+09]];
  CONST robtarget lscs2002838400_B:=[[1425.90,561.62,2171.50],[0.353065,-0.0165687,-0.0612206,-0.933447],[0,-1,0,0],[34.9995,9E+09,9E+09,9E+09,9E+09,9E+09]];
  CONST robtarget lsdcd002932302:=[[2114.43,669.26,2160.75],[0.602613,-0.0234179,-0.0200024,-0.797439],[0,-1,0,0],[35.0003,9E+09,9E+09,9E+09,9E+09,9E+09]];
  CONST robtarget lsdc1002933000:=[[2840.85,-655.82,2169.55],[0.815226,4.73965E-06,6.69998E-06,-0.579144],[0,-1,0,0],[40.0003,9E+09,9E+09,9E+09,9E+09,9E+09]];
  CONST robtarget lsdcg002932401:=[[2250.65,-653.32,2172.05],[0.713307,-2.71637E-06,-1.02355E-05,-0.700852],[0,-1,0,0],[40.2542,9E+09,9E+09,9E+09,9E+09,9E+09]];
  CONST robtarget lsdcg002932301:=[[2114.88,-655.48,2171.91],[0.693602,0.00906872,0.00869882,-0.720249],[0,0,0,0],[35.1918,9E+09,9E+09,9E+09,9E+09,9E+09]];
  CONST robtarget lscs2002947600:=[[2805.89,666.43,2158.90],[0.930861,-0.00993263,-0.0137045,-0.364983],[0,0,-1,0],[35.0002,9E+09,9E+09,9E+09,9E+09,9E+09]];
  CONST robtarget lspac002880400:=[[1516.75,-714.55,1973.69],[0.804938,0.012486,-0.00353793,-0.593217],[-1,0,-1,0],[42.677,9E+09,9E+09,9E+09,9E+09,9E+09]];
  CONST robtarget lspac002880300:=[[1421.05,393.39,1985.45],[0.913275,0.0453431,0.0156622,-0.404509],[-1,-1,-1,0],[29.9928,9E+09,9E+09,9E+09,9E+09,9E+09]];
  CONST robtarget lspac002880200:=[[1421.91,282.35,1989.87],[0.896672,0.029195,0.0199331,-0.441283],[-1,-1,-1,0],[29.9987,9E+09,9E+09,9E+09,9E+09,9E+09]];
  CONST robtarget lspac002880100:=[[1422.03,168.64,1993.18],[0.856739,0.0114723,-0.00538132,-0.515595],[-1,0,-1,0],[29.9999,9E+09,9E+09,9E+09,9E+09,9E+09]];
  CONST robtarget lspac002880000:=[[1422.96,54.80,1994.89],[0.856191,0.0114756,-0.00536636,-0.516505],[-1,0,-1,0],[29.9954,9E+09,9E+09,9E+09,9E+09,9E+09]];
  CONST robtarget lspac002879900:=[[1421.41,-58.39,1996.27],[0.851131,0.0115247,-0.00525309,-0.5248],[-1,0,-1,0],[30.0011,9E+09,9E+09,9E+09,9E+09,9E+09]];
  CONST robtarget lspac002879800:=[[1421.64,-171.93,1997.02],[0.846373,0.0115705,-0.00514874,-0.53244],[-1,0,-1,0],[29.9987,9E+09,9E+09,9E+09,9E+09,9E+09]];
  CONST robtarget lspac002879700:=[[1420.12,-289.05,1997.30],[0.842141,0.0116146,-0.00505557,-0.539109],[-1,0,-1,0],[29.9992,9E+09,9E+09,9E+09,9E+09,9E+09]];
  CONST robtarget lspac002879600:=[[1421.74,-400.76,1992.86],[0.831856,0.0117096,-0.00482765,-0.554848],[-1,0,-1,0],[29.998,9E+09,9E+09,9E+09,9E+09,9E+09]];
  CONST robtarget lspac002879500:=[[1421.14,-513.56,1989.40],[0.820939,0.0118183,-0.00458971,-0.570875],[-1,0,-1,0],[29.9967,9E+09,9E+09,9E+09,9E+09,9E+09]];
  CONST robtarget lscs1002847500:=[[1423.19,-641.19,1984.85],[0.808945,0.0119184,-0.00433887,-0.587747],[-1,0,-1,0],[29.9975,9E+09,9E+09,9E+09,9E+09,9E+09]];
  CONST robtarget lscs1002858300:=[[1424.06,-653.97,1984.84],[0.808291,0.0119288,-0.00431925,-0.588646],[-1,0,-1,0],[29.9978,9E+09,9E+09,9E+09,9E+09,9E+09]];
  CONST robtarget lscs2003266600_1:=[[2778.59,-713.93,1972.36],[0.785632,0.00453952,-0.00354824,-0.618667],[0,0,0,0],[29.9999,9E+09,9E+09,9E+09,9E+09,9E+09]];
  CONST robtarget lscs1002947400_1:=[[3014.96,-658.33,2172.04],[0.825567,0.00172075,0.00251365,-0.564296],[0,-1,0,0],[35.0012,9E+09,9E+09,9E+09,9E+09,9E+09]];
  CONST robtarget lscs2002947700_1:=[[2986.67,662.91,2157.14],[0.961004,1.25775E-05,3.51678E-06,-0.276535],[0,-1,-1,0],[34.9988,9E+09,9E+09,9E+09,9E+09,9E+09]];

  !
  !-----------------------
  !---------XDF-----------
  !-----------------------
  !T_K0_XDF_L2H1
  !-----------------------
  !
  !Robtargets XDF
  CONST robtarget deb_SR2_K0_XD_L2H1:=[[1204.98,540.24,1880.24],[0.834987,0.009454,-0.025984,-0.549575],[-1,0,-1,0],[180,9E+09,9E+09,9E+09,9E+09,9E+09]];
  CONST robtarget SCSCD009469:=[[563.22,371.79,1828.78],[0.627988,0.198147,-0.244598,-0.711717],[-1,0,-1,0],[20,9E+09,9E+09,9E+09,9E+09,9E+09]];
  CONST robtarget SCSCD009472:=[[576.11,455.19,1826.99],[0.625237,0.190136,-0.251531,-0.713904],[-1,0,-1,0],[20,9E+09,9E+09,9E+09,9E+09,9E+09]];

  CONST robtarget SCSDD010167:=[[1428.9,-605.41,1985.83],[0.824974,0.024684,0.005173,-0.564607],[-1,0,-1,0],[10,9E+09,9E+09,9E+09,9E+09,9E+09]];
  CONST robtarget SCSDD010165:=[[1325,-605.41,1985.8],[0.7998,0.016217,0.015589,-0.599845],[-1,-1,-1,0],[10,9E+09,9E+09,9E+09,9E+09,9E+09]];
  CONST robtarget SCSCD010317:=[[1327,-566.9,1988.99],[0.81022,0.011832,0.00518,-0.585984],[-1,-1,-1,0],[10,9E+09,9E+09,9E+09,9E+09,9E+09]];
  CONST robtarget SCSCD010318:=[[1327,-470.2,1992.58],[0.810193,0.014338,0.010366,-0.585897],[-1,-1,-1,0],[10,9E+09,9E+09,9E+09,9E+09,9E+09]];
  CONST robtarget SCSCD010331:=[[1326.97,-448.69,1992.58],[0.808903,0.015416,0.009241,-0.587667],[-1,-1,-1,0],[10,9E+09,9E+09,9E+09,9E+09,9E+09]];
  CONST robtarget SCSCD010319:=[[1327,-340.2,1997.09],[0.814,0.015495,0.009106,-0.580587],[-1,-1,-1,0],[10,9E+09,9E+09,9E+09,9E+09,9E+09]];
  CONST robtarget SCSCD010320:=[[1327,-226.8,1998.62],[0.830219,0.006676,0.004484,-0.557379],[-1,-1,-1,0],[10,9E+09,9E+09,9E+09,9E+09,9E+09]];
  CONST robtarget SCSCD010321:=[[1327,-113.4,2000.01],[0.830234,0.004006,0.002691,-0.557393],[-1,-1,-1,0],[10,9E+09,9E+09,9E+09,9E+09,9E+09]];
  CONST robtarget SCSCD010322:=[[1327.2,16.6,2000.47],[0.830251,-0.001335,-0.000896,-0.557387],[-1,0,-1,0],[10,9E+09,9E+09,9E+09,9E+09,9E+09]];
  CONST robtarget SCSCD010310:=[[1327,113.4,2000.01],[0.830245,-0.004007,-0.002689,-0.557378],[-1,0,-1,0],[10,9E+09,9E+09,9E+09,9E+09,9E+09]];
  CONST robtarget SCSCD010311:=[[1327,226.8,1998.62],[0.843587,-0.006785,-0.004318,-0.536933],[-1,0,-1,0],[10,9E+09,9E+09,9E+09,9E+09,9E+09]];
  CONST robtarget SCSCD010312:=[[1327,340.2,1997.09],[0.848444,0.005278,-0.015155,-0.529041],[-1,0,-1,0],[10,9E+09,9E+09,9E+09,9E+09,9E+09]];
  CONST robtarget SCSCD010330:=[[1326.55,448.23,1993.26],[0.852642,0.000689,-0.017535,-0.5222],[-1,0,-1,0],[10,9E+09,9E+09,9E+09,9E+09,9E+09]];
  CONST robtarget SCSCD010313:=[[1327,470.2,1992.58],[0.849024,-0.015023,-0.009346,-0.528058],[-1,0,-1,0],[10,9E+09,9E+09,9E+09,9E+09,9E+09]];
  CONST robtarget SCSCD010314:=[[1327,566.89,1988.99],[0.862454,-0.018035,-0.010578,-0.505704],[-1,0,-1,0],[10,9E+09,9E+09,9E+09,9E+09,9E+09]];
  CONST robtarget SCSDD010166:=[[1325,605.4,1985.81],[0.866795,-0.019963,-0.010541,-0.498153],[-1,0,-1,0],[10,9E+09,9E+09,9E+09,9E+09,9E+09]];


  !-----------------------
  !T_K0_XDF_L2H2
  !-----------------------

  CONST robtarget SCS2D035686_L2H2:=[[1291.5,556.1,2145.57],[0.302046,0.043202,-0.035344,-0.951658],[0,0,0,0],[10,9E+09,9E+09,9E+09,9E+09,9E+09]];
  CONST robtarget SCSCD009431_L2H2:=[[1291.42,445.69,2150.14],[0.323015,0.047688,-0.032993,-0.944616],[0,0,0,0],[10,9E+09,9E+09,9E+09,9E+09,9E+09]];
  CONST robtarget SCSCD009433_L2H2:=[[1290.8,72.7,2157.07],[0.444271,0.053891,-0.028481,-0.893817],[0,0,0,0],[10,9E+09,9E+09,9E+09,9E+09,9E+09]];
  CONST robtarget SCSCD009430_L2H2:=[[1290.8,-72.8,2157.07],[0.467961,0.055135,-0.023781,-0.881707],[0,0,0,0],[10,9E+09,9E+09,9E+09,9E+09,9E+09]];
  CONST robtarget SCSCD009432_L2H2:=[[1291.61,-448.3,2150.11],[0.525228,0.059117,-0.016951,-0.848736],[-1,0,0,0],[10,9E+09,9E+09,9E+09,9E+09,9E+09]];
  CONST robtarget SCS1D035684_L2H2:=[[1291.5,-556.1,2145.49],[0.540273,0.055438,-0.013487,-0.839553],[-1,0,0,0],[10,9E+09,9E+09,9E+09,9E+09,9E+09]];

  CONST robtarget SCS2D011236_L2H2:=[[2235.4,598.9,2176.97],[0.682904,-0.012195,-0.018,-0.730184],[0,-1,0,0],[20,9E+09,9E+09,9E+09,9E+09,9E+09]];
  CONST robtarget SCSCD009371_L2H2:=[[2230.9,575.4,2179.6],[0.682921,-0.011377,-0.01825,-0.730175],[0,-1,0,0],[20,9E+09,9E+09,9E+09,9E+09,9E+09]];
  CONST robtarget SCSCD009369_L2H2:=[[2135,574.5,2178.74],[0.682974,-0.009192,-0.016852,-0.730191],[0,-1,0,0],[20,9E+09,9E+09,9E+09,9E+09,9E+09]];
  CONST robtarget SCS2D011237_L2H2:=[[2130.3,599.1,2176.19],[0.682892,-0.012768,-0.018144,-0.730182],[0,-1,0,0],[20,9E+09,9E+09,9E+09,9E+09,9E+09]];
  CONST robtarget SCSCD009480_L2H2:=[[1291.71,-509.8,2148.8],[0.511852,0.063343,-0.028455,-0.85623],[-1,0,0,0],[20,9E+09,9E+09,9E+09,9E+09,9E+09]];
  CONST robtarget SCSCD009487_L2H2:=[[1291.21,-382.4,2152.82],[0.51217,0.059721,-0.028917,-0.856317],[-1,0,0,0],[20,9E+09,9E+09,9E+09,9E+09,9E+09]];
  CONST robtarget SCSCD009486_L2H2:=[[1290.91,-254.9,2155.69],[0.500812,0.055499,-0.023021,-0.863468],[0,0,0,0],[20,9E+09,9E+09,9E+09,9E+09,9E+09]];
  CONST robtarget SCSCD009485_L2H2:=[[1290.8,-127.5,2157.46],[0.500481,0.056483,-0.028187,-0.863443],[0,0,0,0],[20,9E+09,9E+09,9E+09,9E+09,9E+09]];
  CONST robtarget SCSCD009482_L2H2:=[[1290.71,-18,2158.03],[0.469882,0.054125,-0.032595,-0.880465],[0,0,0,0],[20,9E+09,9E+09,9E+09,9E+09,9E+09]];
  CONST robtarget SCSCD009481_L2H2:=[[1290.8,127.4,2157.46],[0.469781,0.051291,-0.036782,-0.880524],[0,0,0,0],[20,9E+09,9E+09,9E+09,9E+09,9E+09]];
  CONST robtarget SCSCD009483_L2H2:=[[1290.91,254.69,2155.7],[0.430492,0.048026,-0.034121,-0.90067],[0,0,0,0],[20,9E+09,9E+09,9E+09,9E+09,9E+09]];
  CONST robtarget SCSCD009484_L2H2:=[[1291.21,382.12,2152.79],[0.355613,0.05454,-0.0411734,-0.932132],[0,0,0,0],[20.0032,9E+09,9E+09,9E+09,9E+09,9E+09]];
  CONST robtarget SCSCD009477_L2H2:=[[1291.48,509.42,2148.80],[0.300043,0.0559945,-0.0394357,-0.951464],[0,0,0,0],[19.9993,9E+09,9E+09,9E+09,9E+09,9E+09]];
  CONST robtarget SCSCD009478_L2H2:=[[1292.91,648.49,2143.94],[0.276939,0.042757,-0.038699,-0.959155],[0,0,0,0],[20,9E+09,9E+09,9E+09,9E+09,9E+09]];
  CONST robtarget SCS2D010234_L2H2:=[[1432.5,700.1,2143.82],[0.282576,0.037813,-0.032439,-0.95795],[0,0,0,0],[20,9E+09,9E+09,9E+09,9E+09,9E+09]];
  CONST robtarget SCSCD009429_L2H2:=[[1395.3,160,2167.49],[0.500685,0.033709,-0.02751,-0.864535],[0,0,0,0],[20,9E+09,9E+09,9E+09,9E+09,9E+09]];
  CONST robtarget SCSCD009427_L2H2:=[[1395.2,47,2168.33],[0.501,0.036953,-0.02238,-0.864368],[0,0,0,0],[20,9E+09,9E+09,9E+09,9E+09,9E+09]];
  CONST robtarget SCSCD009434_L2H2:=[[1395.2,-47,2168.29],[0.501038,0.035952,-0.021969,-0.864399],[0,0,0,0],[20,9E+09,9E+09,9E+09,9E+09,9E+09]];
  CONST robtarget SCSCD009428_L2H2:=[[1395.31,-160,2167.42],[0.501234,0.043522,-0.017169,-0.864046],[0,0,0,0],[20,9E+09,9E+09,9E+09,9E+09,9E+09]];
  CONST robtarget SCSCD009422_L2H2:=[[1395.52,-260.8,2165.81],[0.501356,0.045052,-0.014502,-0.863946],[0,0,0,0],[20,9E+09,9E+09,9E+09,9E+09,9E+09]];
  CONST robtarget SCSCD009421_L2H2:=[[1395.72,-361.7,2163.61],[0.501496,0.047087,-0.011035,-0.863807],[0,0,0,0],[20,9E+09,9E+09,9E+09,9E+09,9E+09]];
  CONST robtarget SCSCD009426_L2H2:=[[1396,-462.5,2160.76],[0.501522,0.047531,-0.010336,-0.863777],[0,0,0,0],[20,9E+09,9E+09,9E+09,9E+09,9E+09]];
  CONST robtarget SCS1D035683_L2H2_:=[[1395,-564.9,2155.92],[0.501271,0.042073,-0.016812,-0.864103],[0,0,0,0],[20,9E+09,9E+09,9E+09,9E+09,9E+09]];
  CONST robtarget SCS1D009539_L2H2:=[[1476.81,-697.79,2148.77],[0.569434,0.041061,0.009952,-0.820951],[0,0,0,0],[20,9E+09,9E+09,9E+09,9E+09,9E+09]];
  CONST robtarget SCS1D009551_L2H2:=[[1536.9,-700.9,2151.19],[0.569657,0.032461,0.007702,-0.821205],[0,0,0,0],[20,9E+09,9E+09,9E+09,9E+09,9E+09]];
  CONST robtarget SCS1D009540_L2H2:=[[1628.7,-700.5,2154.83],[0.569981,0.027085,0.011218,-0.821135],[0,0,0,0],[20,9E+09,9E+09,9E+09,9E+09,9E+09]];
  CONST robtarget SCS1D009541_L2H2:=[[1720.7,-700.3,2157.37],[0.57018,0.023843,0.013434,-0.821064],[0,0,0,0],[20,9E+09,9E+09,9E+09,9E+09,9E+09]];
  CONST robtarget SCS1D009542_L2H2:=[[1812.62,-700.09,2159.27],[0.562278,0.0209611,0.0160003,-0.826528],[0,0,0,0],[19.9996,9E+09,9E+09,9E+09,9E+09,9E+09]];
  CONST robtarget SCSCD009372_L2H2:=[[2134.5,-460.5,2182.98],[0.587566,0.013497,0.00984,-0.809003],[0,0,0,0],[20,9E+09,9E+09,9E+09,9E+09,9E+09]];
  CONST robtarget SCSCD009361_L2H2:=[[2134.8,-369.2,2185.69],[0.587594,0.011442,0.0079,-0.809036],[0,0,0,0],[20,9E+09,9E+09,9E+09,9E+09,9E+09]];
  CONST robtarget SCSCD009374_L2H2:=[[2135,-205.7,2188.94],[0.587633,0.008109,0.003253,-0.80908],[0,0,0,0],[20,9E+09,9E+09,9E+09,9E+09,9E+09]];
  CONST robtarget SCSCD009373_L2H2:=[[2135.8,-14.5,2190.55],[0.587632,0.004571,-0.002417,-0.809111],[0,0,0,0],[20,9E+09,9E+09,9E+09,9E+09,9E+09]];
  CONST robtarget SCSCD009363_L2H2:=[[2230.9,0,2191.4],[0.643317,0.003297,-0.001961,-0.76559],[0,0,0,0],[20,9E+09,9E+09,9E+09,9E+09,9E+09]];
  CONST robtarget SCSCD009362_L2H2:=[[2230.9,-163,2190.44],[0.601663,0.007154,0.003863,-0.798708],[0,0,0,0],[20,9E+09,9E+09,9E+09,9E+09,9E+09]];
  CONST robtarget SCSCD009370_L2H2:=[[2230.9,-248.6,2189.18],[0.587637,0.003427,-0.001724,-0.809116],[0,0,0,0],[20,9E+09,9E+09,9E+09,9E+09,9E+09]];
  CONST robtarget SCSCD009360_L2H2:=[[2230.9,-417.5,2185.13],[0.62915,0.012822,0.009604,-0.777119],[0,0,0,0],[20,9E+09,9E+09,9E+09,9E+09,9E+09]];
  CONST robtarget SCSCD009358_L2H2:=[[2230.9,-575.4,2179.6],[0.66891,0.017208,0.0129,-0.743032],[0,0,0,0],[20,9E+09,9E+09,9E+09,9E+09,9E+09]];
  CONST robtarget SCS1D011234_L2H2:=[[2235.4,-598.9,2176.97],[0.706883,0.017586,0.012787,-0.706997],[0,0,0,0],[20,9E+09,9E+09,9E+09,9E+09,9E+09]];
  CONST robtarget SCS1D009546_L2H2:=[[2183.8,-697.2,2163.51],[0.706829,0.020657,0.014551,-0.706933],[0,0,0,0],[20,9E+09,9E+09,9E+09,9E+09,9E+09]];
  CONST robtarget SCS1D009547_L2H2:=[[2278.4,-699.5,2164.85],[0.706836,0.020007,0.015201,-0.706931],[0,0,0,0],[20,9E+09,9E+09,9E+09,9E+09,9E+09]];
  CONST robtarget SCS1D009548_L2H2:=[[2405.8,-699.4,2165.58],[0.706863,0.018417,0.014655,-0.706959],[0,0,0,0],[20,9E+09,9E+09,9E+09,9E+09,9E+09]];
  CONST robtarget SCS1D009549_L2H2:=[[2533.1,-699.3,2166.28],[0.706838,0.01937,0.016311,-0.706922],[0,0,0,0],[20,9E+09,9E+09,9E+09,9E+09,9E+09]];
  CONST robtarget SCS1D009553_L2H2:=[[2660.4,-699.3,2166.72],[0.742857,0.020657,0.016812,-0.66892],[0,0,0,0],[20,9E+09,9E+09,9E+09,9E+09,9E+09]];
  CONST robtarget SCS1D009552_L2H2:=[[2787.7,-699.2,2167.07],[0.725092,0.02021,0.017347,-0.688137],[0,0,0,0],[20,9E+09,9E+09,9E+09,9E+09,9E+09]];
  CONST robtarget SCS1D009927_L2H2:=[[3009.3,-698.7,2168.15],[0.793095,0.02015,0.014943,-0.608581],[0,0,0,0],[20,9E+09,9E+09,9E+09,9E+09,9E+09]];
  CONST robtarget SCSCD009418_L2H2:=[[2957.3,-623.6,2180.39],[0.818762,0.018267,0.013513,-0.573683],[0,0,0,0],[20,9E+09,9E+09,9E+09,9E+09,9E+09]];
  CONST robtarget SCSCD009400_L2H2:=[[2957.30,-570.30,2182.67],[0.813058,-0.0188169,-0.0127276,-0.581739],[0,-1,0,0],[20.0002,9E+09,9E+09,9E+09,9E+09,9E+09]];
  CONST robtarget SCSCD009398_L2H2:=[[2957.30,-456.29,2186.85],[0.813774,0.0123654,0.00960675,-0.580971],[0,0,0,0],[19.9996,9E+09,9E+09,9E+09,9E+09,9E+09]];
  CONST robtarget SCSCD009408_L2H2:=[[2957.39,-342.30,2190.10],[0.824026,0.0113569,0.00739682,-0.566389],[0,0,0,0],[19.9999,9E+09,9E+09,9E+09,9E+09,9E+09]];
  CONST robtarget SCSCD009416_L2H2:=[[2957.39,-228.20,2192.36],[0.832467,0.0061603,0.00442599,-0.554023],[0,0,0,0],[19.9999,9E+09,9E+09,9E+09,9E+09,9E+09]];
  CONST robtarget SCSCD009406_L2H2:=[[2957.50,-114.10,2193.77],[0.836429,0.00377205,0.00248688,-0.548057],[0,-1,0,0],[20.0002,9E+09,9E+09,9E+09,9E+09,9E+09]];
  CONST robtarget SCSCD009414_L2H2:=[[2957.49,-17.99,2194.23],[0.839284,0.00208987,0.00278511,-0.543682],[0,-1,0,0],[19.9999,9E+09,9E+09,9E+09,9E+09,9E+09]];
  CONST robtarget SCSCD009404_L2H2:=[[2957.50,114.11,2193.76],[0.858392,-0.00375915,-0.00250521,-0.512974],[0,-1,-1,0],[19.9999,9E+09,9E+09,9E+09,9E+09,9E+09]];
  CONST robtarget SCSCD009412_L2H2:=[[2957.4,228.2,2192.35],[0.866848,-0.00595,-0.002347,-0.498531],[0,-1,-1,0],[20,9E+09,9E+09,9E+09,9E+09,9E+09]];
  CONST robtarget SCSCD009410_L2H2:=[[2957.4,342.3,2190.1],[0.895222,-0.011834,-0.006628,-0.445414],[0,-1,-1,0],[20,9E+09,9E+09,9E+09,9E+09,9E+09]];
  CONST robtarget SCSCD009396_L2H2:=[[2957.3,456.3,2186.8],[0.92033,-0.014333,-0.01209,-0.390692],[0,-1,-1,0],[20,9E+09,9E+09,9E+09,9E+09,9E+09]];
  CONST robtarget SCSCD009402_L2H2:=[[2957.3,570.3,2182.66],[0.942168,-0.01884,-0.005547,-0.334564],[0,-1,-1,0],[20,9E+09,9E+09,9E+09,9E+09,9E+09]];
  CONST robtarget SCSCD009420_L2H2:=[[2957.3,623.6,2180.39],[0.942107,-0.021601,-0.007036,-0.334541],[0,-1,-1,0],[20,9E+09,9E+09,9E+09,9E+09,9E+09]];
  CONST robtarget SCSCD009382_L2H2:=[[3062.4,575.4,2182.56],[0.819161,-0.016688,-0.012133,-0.573192],[0,-1,0,0],[20,9E+09,9E+09,9E+09,9E+09,9E+09]];
  CONST robtarget SCSCD009384_L2H2:=[[3062.4,432.3,2186.93],[0.819161,-0.016688,-0.012133,-0.573192],[0,-1,0,0],[20,9E+09,9E+09,9E+09,9E+09,9E+09]];
  CONST robtarget SCSCD009394_L2H2:=[[3062.4,288.2,2190.66],[0.819193,-0.008634,-0.004077,-0.573439],[0,-1,0,0],[20,9E+09,9E+09,9E+09,9E+09,9E+09]];
  CONST robtarget SCSCD009378_L2H2:=[[3062.4,144.1,2192.89],[0.819052,-0.002561,-0.004706,-0.573695],[0,-1,0,0],[20,9E+09,9E+09,9E+09,9E+09,9E+09]];
  CONST robtarget SCSCD009386_L2H2:=[[3062.4,0,2193.65],[0.819091,-0.001733,-0.001707,-0.573658],[0,-1,0,0],[20,9E+09,9E+09,9E+09,9E+09,9E+09]];
  CONST robtarget SCSCD009380_L2H2:=[[3062.4,-144.1,2192.86],[0.819102,0.002709,0.007554,-0.573592],[0,-1,0,0],[20,9E+09,9E+09,9E+09,9E+09,9E+09]];
  CONST robtarget SCSCD009392_L2H2:=[[3062.4,-288.2,2190.6],[0.818916,0.010102,0.005,-0.573803],[0,0,0,0],[20,9E+09,9E+09,9E+09,9E+09,9E+09]];
  CONST robtarget SCSCD009388_L2H2:=[[3062.4,-432.3,2186.88],[0.818839,0.014036,0.006838,-0.573811],[0,0,0,0],[20,9E+09,9E+09,9E+09,9E+09,9E+09]];
  CONST robtarget SCSCD009390_L2H2:=[[3062.42,-574.45,2181.74],[0.818814,0.01631,0.013203,-0.573676],[0,0,0,0],[80,9E+09,9E+09,9E+09,9E+09,9E+09]];
  CONST robtarget SCSGD010159_L2H2:=[[3062.4,-646.9,2179.4],[0.818747,0.019042,0.012903,-0.573693],[0,0,0,0],[80,9E+09,9E+09,9E+09,9E+09,9E+09]];
  CONST robtarget SCS1D010180_L2H2:=[[3105,-697.4,2168.29],[0.81871,0.020581,0.013931,-0.573669],[0,0,0,0],[20,9E+09,9E+09,9E+09,9E+09,9E+09]];

  CONST robtarget SCS1D009550_L2H2:=[[2915.1,-699.2,2167.3],[0.793075,0.020945,0.014995,-0.608579],[0,0,0,0],[20,9E+09,9E+09,9E+09,9E+09,9E+09]];
  CONST robtarget SCSCD009359_L2H2:=[[2136.2,-574.5,2178.75],[0.710017,0.016561,0.009662,-0.703923],[0,0,0,0],[20,9E+09,9E+09,9E+09,9E+09,9E+09]];
  CONST robtarget SCS1D011235_L2H2:=[[2130.3,-599.1,2176.19],[0.706842,0.017705,0.01337,-0.707024],[0,0,0,0],[20,9E+09,9E+09,9E+09,9E+09,9E+09]];
  CONST robtarget SCS1D009545_L2H2:=[[2088.5,-699.7,2163.18],[0.684266,0.021012,0.014434,-0.728787],[0,0,0,0],[20,9E+09,9E+09,9E+09,9E+09,9E+09]];
  CONST robtarget SCS1D009544_L2H2:=[[1996.6,-699.8,2162.12],[0.657704,0.022745,0.015338,-0.752777],[0,0,0,0],[20,9E+09,9E+09,9E+09,9E+09,9E+09]];
  CONST robtarget SCS1D009543_L2H2:=[[1904.6,-699.9,2160.87],[0.633077,0.021073,0.01446,-0.773667],[0,0,0,0],[20,9E+09,9E+09,9E+09,9E+09,9E+09]];

  !========================
  ! Calcul de code interne
  !========================
  LOCAL FUNC num Code_Interne()
    ! Calculer le code a executer
    ! en fonction des conditions
    ! internes et retourner
    ! le code calcule
    !
    ! Ex: return XXX
    ! Si pas de code interne
    RETURN 0;
  ENDFUNC

  !=======================
  ! Gestion des programmes
  !=======================
  PROC Programme(
    num prog)

  	!Option Securité
		IF EPSRequest THEN
			AutoriseTraj;
			T_TrajSYNC;
		ENDIF
		!
    TEST prog
    CASE 21:
      Aff_Prog prog,"X62E1H1";
      ! pulse sur la sortie Acquittement code
      PulseDO\PLength:=1,ACQ_CODE1;
      AutoriseTraj;
      T_X62E1H1;
    CASE 23:
      Aff_Prog prog,"X62E2H2";
      ! pulse sur la sortie Acquittement code
      PulseDO\PLength:=1,ACQ_CODE1;
      AutoriseTraj;
      T_X62E2H2;
    CASE 25:
      Aff_Prog prog,"X62E3H2";
      ! pulse sur la sortie Acquittement code
      PulseDO\PLength:=1,ACQ_CODE1;
      AutoriseTraj;
      T_X62E3H2;
    CASE 26:
      Aff_Prog prog,"X62CC";
      ! pulse sur la sortie Acquittement code
      PulseDO\PLength:=1,ACQ_CODE1;
      AutoriseTraj;
      T_X62CC;
    CASE 27:
      Aff_Prog prog,"X62E3H2B";
      ! pulse sur la sortie Acquittement code
      PulseDO\PLength:=1,ACQ_CODE1;
      AutoriseTraj;
      T_X62E3H2B;
    CASE 53:
      Aff_Prog prog,"T_CHELM_P1";
      ! pulse sur la sortie Acquittement code
      PulseDO\PLength:=1,ACQ_CODE1;
      AutoriseTraj;
      T_CHELM_P1;
      !
      !MOD AMBULANCIA
      !
    CASE 30:
      Aff_Prog prog,"T_XDF_L2H1";
      ! pulse sur la sortie Acquittement code
      PulseDO\PLength:=1,ACQ_CODE1;
      AutoriseTraj;
      !T_XDF_L2H1;
    CASE 31:
      Aff_Prog prog,"T_XDF_L2H2";
      ! pulse sur la sortie Acquittement code
      PulseDO\PLength:=1,ACQ_CODE1;
      AutoriseTraj;
      T_XDF_L2H2;
      !
    CASE 124:
      Aff_Prog prog,"X62E1H1AMB";
      ! pulse sur la sortie Acquittement code
      PulseDO\PLength:=1,ACQ_CODE1;
      AutoriseTraj;
      T_X62E1H1;
    CASE 125:
      Aff_Prog prog,"X62E2H2AMB";
      ! pulse sur la sortie Acquittement code
      PulseDO\PLength:=1,ACQ_CODE1;
      AutoriseTraj;
      T_X62E2H2;
    CASE 126:
      Aff_Prog prog,"X62E3H2AMB";
      ! pulse sur la sortie Acquittement code
      PulseDO\PLength:=1,ACQ_CODE1;
      AutoriseTraj;
      T_X62E3H2;
      !
      !Enlever les commentaires pour l'option Changeur Outil
!    CASE 200:
!      Aff_Prog prog,"Chg Toute Electrode";
!      ! pulse sur la sortie Acquittement code
!      PulseDO\PLength:=1,ACQ_CODE1;
!      AutoriseTraj;
!      T_Serv1_ALL;
    !
    ! ne pas modifier la fin de la routine
    !


    CASE CP_CODE_NUL:
      Aff_Prog 0,strEMPTY;
      Aff_Traj strEMPTY;
    DEFAULT:
      Aff_Prog prog,strEMPTY;
      Aff_Traj strEMPTY;
    ENDTEST
  ENDPROC

  !-----------------------
  ! Procédures de Service
  !-----------------------
  PROC Services(
    num sprog)
    TEST sprog
    CASE CP_DemServ1:
      Aff_Prog sprog,"Chg_Elec";
      AutoriseTraj;
      T_Serv1;
      Etat_Serv1:=EtatService1{noThisTask};
    CASE CP_DemServ2:
      Aff_Prog sprog,"Rodage";
      AutoriseTraj;
      T_Serv2;
      Etat_Serv2:=EtatService2{noThisTask};
    CASE CP_DemServ3:
      Aff_Prog sprog,"Verifier";
      AutoriseTraj;
      T_Serv3;
      Etat_Serv3:=SV_PAS_DEMANDE;
    CASE CP_DemServ4:
      Aff_Prog sprog,"Manutencao";
      AutoriseTraj;
      T_Serv4;
      Etat_Serv4:=SV_PAS_DEMANDE;
    DEFAULT:
    ! ajouter par un ERRWRITE
    ENDTEST
  ENDPROC

  PROC PresPrgmvt()
    !******************************
    !*       ATTENTION !!!!!      *
    !*  ROUTINE A NE PAS MODIFIER *
    !*  ET A NE PAS SUPPRIMER !!  *
    !* Utilisé pour test présence *
    !* module PRG_MVT en mémoire  *
    !******************************
  ENDPROC

  PROC LireCodeInterne(
    INOUT num prog)
    !******************************
    !*       ATTENTION !!!!!      *
    !*  ROUTINE A NE PAS MODIFIER *
    !*  ET A NE PAS SUPPRIMER !!  *
    !******************************
    prog:=Code_Interne();
  ENDPROC

  PROC MAIN()
    !******************************
    !*       ATTENTION !!!!!      *
    !*  ROUTINE A NE PAS MODIFIER *
    !*  ET A NE PAS SUPPRIMER !!  *
    !******************************
    LancePromia;
  ENDPROC

  !--------------------------
  ! Trajectoire de lancement
  !--------------------------
  PROC T_Lance()
    Aff_Traj "Lance";
    AntiReboucle;
    !
    MoveJ p_repli,V_moyen,Z_arret,Tool_defaut;
    !
    ! O9:segurança traseira com K1
    ! O12:fora de interferencia1 com K5
    ! O13:fora de interferencia2 com K5
    ORDRE\O9\O12\O13;
    !
    MoveL [[438.93,-1578.56,-395.13],[0.00177362,-0.640935,-0.767576,0.00518556],[-1,-1,0,0],[72.8978,9E+09,9E+09,9E+09,9E+09,9E+09]], V_moyen, Z_moyen, Tool_defaut;
    MoveL [[607.59,-1578.56,937.89],[0.00103662,-0.741078,-0.671396,0.00538228],[-1,-1,0,0],[152.971,9E+09,9E+09,9E+09,9E+09,9E+09]], V_moyen, Z_moyen, Tool_defaut;
    MoveJ p_reb_prg, V_moyen, Z_arret, Tool_defaut;
    !
    T_SEGURANCATRASEIRA;
    !
    SR_INIT_PINCE 1;
    !
  ENDPROC

  !----------------------
  ! Trajectoire de Repli
  !----------------------
  PROC T_Repli()
    Aff_Traj "Repli";
    AntiReboucle;
    !
    MoveJ p_reb_prg,V_moyen,Z_arret,Tool_defaut;
    !
    T_SEGURANCATRASEIRA;
    !
    MoveL [[607.59,-1578.56,937.88],[0.00103673,-0.741078,-0.671396,0.00538257],[-1,-1,0,0],[152.971,9E+09,9E+09,9E+09,9E+09,9E+09]], V_moyen, Z_moyen, Tool_defaut;
    MoveL [[438.93,-1578.56,-395.13],[0.00177362,-0.640935,-0.767576,0.00518556],[-1,-1,0,0],[72.8978,9E+09,9E+09,9E+09,9E+09,9E+09]], V_moyen, Z_moyen, Tool_defaut;
    MoveJ p_repli, V_moyen, Z_arret, Tool_defaut;
    !
    T_SEGURANCATRASEIRA;
    !
  ENDPROC

  !-----------------------------
  ! Trajectoire de Repli direct
  !-----------------------------
  PROC T_Repli_Direct()
    Aff_Traj "Repli direct";
    AntiReboucle;
    MoveJ p_repli,V_lent,Z_arret,Tool_defaut;
  ENDPROC

  !-------------------------
  ! Trajectoires de Service
  !-------------------------
  PROC T_Serv1()
    ! Action param du chgt electodes
    SR_CHG_ELEC\SANS_CHG_1\CHG_DISSOCIE;
    ! ACTION CHGT ELECTRODES
    SR_APPEL_SERV1;
    FOR i FROM 1 TO NbEquipt{noThisTask} DO
      IF SR_APPEL_AUTO(i)=1 OR SR_APPEL_AUTO(i)=2 THEN
        %"T_Chela"+ValToStr(swInRunServ1{noThisTask})%;
        IF SR_APPEL_AUTO(i)=2 THEN
          SR_FIN_SERV1;
          RETURN;
        ENDIF
      ENDIF
      IF SR_APPEL_MANU(i)=1 OR SR_APPEL_MANU(i)=2 THEN
        %"T_Chelm"+ValToStr(swInRunServ1{noThisTask})%;
        IF SR_APPEL_MANU(i)=2 THEN
          SR_FIN_SERV1;
          RETURN;
        ENDIF
      ENDIF
    ENDFOR
    SR_FIN_SERV1;
  ERROR
    IF ERRNO=ERR_CALLPROC OR ERRNO=ERR_REFUNKPRC THEN
      SkipWarn;
      TRYNEXT;
    ENDIF
  ENDPROC

  !-----------------------------------------
  ! Trajectoires de Service Toutes Electrodes
  !-----------------------------------------
  !Enlever les commentaires pour l'option Changeur Outil
!  PROC T_Serv1_ALL()
!    SR_CHG_ELEC\SANS_CHG_1\CHG_DISSOCIE;
!    SR_SERVICE 1\AppelTraj:="T_CHELM_P1"\ChgElect;
!    SR_VALID_CHELMAN;
!    SR_SERVICE 2\AppelTraj:="T_CHELM_P2"\ChgElect;
!    SR_VALID_CHELMAN;
!    SR_SERVICE 3\AppelTraj:="T_CHELM_P3"\ChgElect;
!    SR_VALID_CHELMAN;
!    SR_SERVICE 4\AppelTraj:="T_CHELM_P4"\ChgElect;
!  ENDPROC

  !-------------
  PROC T_Serv2()
    ! Action param du RODAGE
    SR_ROD_ELEC\AVEC_ROD_1\ROD_DISSOCIE;
    ! ACTION RODAGE
    SR_APPEL_SERV2;
    FOR i FROM 1 TO NbEquipt{noThisTask} DO
      IF SR_APPEL_DRESS(i)=1 OR SR_APPEL_DRESS(i)=2 THEN
        %"T_ROD_"+ValToStr(swInRunServ2{noThisTask})%;
        IF SR_APPEL_DRESS(i)=2 THEN
          SR_FIN_SERV2;
          RETURN;
        ENDIF
      ENDIF
    ENDFOR
    SR_FIN_SERV2;
  ERROR
    IF ERRNO=ERR_CALLPROC OR ERRNO=ERR_REFUNKPRC THEN
      SkipWarn;
      TRYNEXT;
    ENDIF
  ENDPROC

  !-------------
  PROC T_Serv3()
    !Chama rotina de verificacao da pinca atual
    AutoriseTraj;
    T_Verificar_P1;
    !
  ENDPROC

  !-------------
  PROC T_Serv4()
    Aff_Traj "Monitoramento";
    AntiReboucle;
    !
    !Servico de Monitoramento das Pincas
    AutoriseTraj;
    T_Monitoramento;
  ENDPROC

  !-----------------------------
  ! Trajectoire de Service SR
  !-----------------------------
  !------------
  !Mettre en commentaires la routine pour l'option Changeur Outil
  PROC T_ROD_1()
    Aff_Traj "T_ROD_1";
    AntiReboucle;
    !
    ! Home Position
    MoveJ p_reb_prg,V_moyen,Z_arret,Tool_defaut;
    !
    AutoriseTraj;
    T_Repli;
    !
    AutoriseTraj;
    T_RODCYCLE_P1;
    !
    AutoriseTraj;
    T_Lance;
    !
  ENDPROC

  !------------
  PROC T_ROD_2()
    Aff_Traj "T_ROD_2";
    AntiReboucle;
    ! Traj rodage Séquenceur 2 pince 2
    MoveJ p_reb_prg,V_moyen,Z_arret,Tool_defaut;
    ! Trajectoire approche
    ! SR_RODER 2,2;
    ! trajectoire dégagement
    SR_INIT_PINCE 0\no_pince2:=2;
    SR_SOUDER p_reb_prg,V_moyen,0,31\no_pince2:=2\prg_soud2:=32,Tool_defaut,wobj0;
  ENDPROC

  !------------
  PROC T_ROD_12()
    Aff_Traj "T_ROD_12";
    AntiReboucle;
    ! Traj rodage séquenceurs 1 et 2 pinces 1 et 2
    MoveJ p_reb_prg,V_moyen,Z_arret,Tool_defaut;
    ! Trajectoire approche
    SR_RODER 1,1;
    ! Trajectoire approche
    SR_RODER 2,2;
    ! trajectoire dégagement
    MoveJ p_reb_prg,V_moyen,Z_arret,Tool_defaut;
    SR_INIT_PINCE 1\no_pince2:=2;
    SR_SOUDER p_reb_prg,V_moyen,1,31\no_pince2:=2\prg_soud2:=32,Tool_defaut,wobj0;
  ENDPROC

  !------------
  !Mettre en commentaires la routine pour l'option Changeur Outil
  PROC T_Chelm1()
    Aff_Traj "T_Chelm1";
    AntiReboucle;
    !
    ! Home Position
    MoveJ p_reb_prg,V_moyen,Z_arret,Tool_defaut;
    !
    AutoriseTraj;
    T_Repli;
    !
    AutoriseTraj;
    T_RODCYCLE_P1;
    !
    ! Trajectoire approche
    MoveJ p_repli, V_moyen, Z_arret, Tool_defaut;
    SR_CEAU 1;
    MoveL pTrocaEletrodosPinca1, V_moyen, Z_arret, Tool_Pince1;
    !
    ! O9:segurança traseira com K1
    ! O12:fora de interferencia1 com K5
    ! O13:fora de interferencia2 com K5
    ! O15:Sinalizacao de Troca de Eletrodo
    ORDRE\O9\O12\O13\O15;
    !
    !E15:autorização de recuo troca de eletrodos pinca 1
    EVENT\E15;
    SR_CHELAUTO 1;
    SR_CEAU 0;
    !
    MoveJ p_repli, V_moyen, Z_arret, Tool_defaut;
    SR_INIT_PINCE 1;
    SR_SOUDER p_repli,V_moyen,1,255,Tool_defaut,wobj0;
    !
    AutoriseTraj;
    T_RODCYCLE_P1;
    !
    AutoriseTraj;
    T_Lance;
    !
  ENDPROC

  !------------
  PROC T_Chelm2()
    Aff_Traj "T_Chelm2";
    AntiReboucle;
    ! Traj chgt manu séquenceur 2 Pince 2
  ENDPROC

  !------------
  PROC T_Chelm12()
    Aff_Traj "T_Chelm12";
    AntiReboucle;
    ! Traj chgt manu séquenceurs 1 et 2 pinces 1 et 2
  ENDPROC

  !------------
  PROC T_Chela1()
    Aff_Traj "T_Chela1";
    AntiReboucle;
    ! Traj chgt auto Tool_Pince 1
    MoveJ p_reb_prg,V_moyen,Z_arret,Tool_defaut;
    !SR_CHANGEUR_AUTO 1\CPPEI\CPPES\SM\OUVRE;
    !Traj Approche Changeur
    SR_CEAU 1;
    !SR_RECAL_PINCE\CORR_ELEC1,[[-49.1,196.04,-129.7],[0.703563,0.00097,-0.000327,-0.710633],[1,-2,-3,1],[109,9E+09,9E+09,9E+09,9E+09,9E+09]],1,V_lent,Z_arret,Tool_Pince1,wobj0;
    !Traj Approche Extracteur
    !MoveL Arret sur point d'extraction
    !SR_CHANGEUR_AUTO 1\SM\FERME;
    !Traj Degagement Extracteur
    !MoveL Arret sur point de controle extraction
    !SR_CHANGEUR_AUTO 1\CPPEI\CPPES\SM\OUVRE;
    !Traj approche Mise
    !MoveL Arret sur point de mise electrode
    !SR_SERRER 1,250,0\Temps:=2;
    !Traj Degagement Mise
    !SR_SERRER 1,250,0\Temps:=2;
    !Traj Approche Extracteur
    !SR_RECAL_PINCE\CORR_ELEC2,[[-49.1,196.04,-129.7],[0.703563,0.00097,-0.000327,-0.710633],[1,-2,-3,1],[109,9E+09,9E+09,9E+09,9E+09,9E+09]],1,V_lent,Z_arret,Tool_Pince1,wobj0;
    !MoveL Arret sur point d'extraction
    !SR_CHANGEUR_AUTO 1\SM\FERME;
    !Traj Degagement Extracteur
    !MoveL Arret sur point de controle extraction
    !SR_CHANGEUR_AUTO 1\CPPEI\CPPES\SM\OUVRE;
    !Traj approche Mise
    !MoveL Arret sur point de mise electrode
    !SR_SERRER 1,250,0\Temps:=2;
    !Traj Degagement Mise
    !SR_RECAL_PINCE\SANS_CORR,[[-49.1,196.04,-129.7],[0.703563,0.00097,-0.000327,-0.710633],[1,-2,-3,1],[109,9E+09,9E+09,9E+09,9E+09,9E+09]],1,V_lent,Z_arret,Tool_Pince1,wobj0;
    !SR_SERRER 1,250,0\Temps:=2;
    !SR_CHELAUTO 1;
    !SR_CEAU 0;
    ! trajectoire dégagement
    MoveJ p_reb_prg,V_moyen,Z_arret,Tool_defaut;
    SR_INIT_PINCE 1;
    SR_SOUDER p_reb_prg,V_moyen,1,31,Tool_defaut,wobj0;
  ENDPROC

  !------------
  PROC T_Chela2()
    Aff_Traj "T_Chela2";
    AntiReboucle;
    ! Traj chgt auto séquenceurs 2 pince 2
  ENDPROC

  !------------
  PROC T_Chela12()
    Aff_Traj "T_Chela12";
    AntiReboucle;
    ! Traj chgt auto séquenceurs 1 et 2 pinces 1 et 2
  ENDPROC

  !------------
  PROC T_Verificar_P1()
    Aff_Traj "T_Verificar_P1";
    AntiReboucle;
    !
    !Home Position
    MoveJ p_reb_prg,V_moyen,Z_arret,Tool_defaut;
    !
    AutoriseTraj;
    T_Repli;
    !
    ! Traj Verificacao Pinca 1
    MoveJ p_repli, V_moyen, Z_arret, Tool_defaut;
    MoveJ [[117.15,-2672.79,-820.13],[0.578822,-0.00575543,0.000189017,-0.815433],[-1,-1,0,0],[72.8969,9E+09,9E+09,9E+09,9E+09,9E+09]], V_moyen, Z_Xlarge, Tool_Pince1;
    MoveL pReferenciaPinca1, V_lent, Z_arret, Tool_Pince1;
    !
    T_Mensagem;
    !
    MoveL [[117.15,-2672.79,-820.13],[0.578822,-0.00575565,0.000188069,-0.815433],[-1,-1,0,0],[72.8966,9E+09,9E+09,9E+09,9E+09,9E+09]], V_lent, Z_Xlarge, Tool_Pince1;
    MoveL [[615.94,-2670.60,-863.81],[0.761828,-0.00559545,0.00156093,-0.647753],[-1,-1,0,0],[72.8897,9E+09,9E+09,9E+09,9E+09,9E+09]], V_lent, Z_Xlarge, Tool_Pince1;
    MoveJ p_repli, V_moyen, Z_arret, Tool_defaut;
    !
    AutoriseTraj;
    T_Lance;
    !
  ENDPROC

	!-----------
	PROC T_Mensagem()
		!
		VAR btnres btnMensagem:=0;
		VAR string strMensagem {7}:=[
		"Vire a chave para FS (Fora de servico).",
		"Abra a porta da celula.",
		"Verifique a ferramenta.",
		"Apos a verificacao, feche a porta.",
		"Vire a chave para ES (Em Servico)",
		"Pressione o botao MARCHA CICLO no painel.",
		"Pressione OK abaixo para confirmar."];
		!
		btnMensagem := UIMessageBox(\Header:="       Verificacao de Ferramenta"\MsgArray:=strMensagem\Buttons:=btnOK\Icon:=iconInfo);
  ENDPROC

  !------------
  !Option Securité
  PROC T_TrajSYNC()
  	!
		Aff_Traj "TrajSYNC";
		AntiReboucle;
		!
    !
    !Home Position
    MoveJ p_reb_prg,V_moyen,Z_arret,Tool_defaut;
    !
    AutoriseTraj;
    T_Repli;
    !
    MoveJ p_repli, V_moyen, Z_arret, Tool_defaut;
    MoveJ [[482.36,-1628.63,-396.89],[0.000391776,-0.815436,-0.578822,0.00546986],[-1,-1,0,0],[72.8969,9E+09,9E+09,9E+09,9E+09,9E+09]], V_moyen, Z_Xlarge, Tool_defaut;
    MoveAbsJ pPSync,V_moyen,Z_arret,Tool_defaut;
    !
    SoftwareSync;
    IF diEPS_Sync =1 EPSRequest:=FALSE;
    !
    MoveL [[482.36,-1628.63,-396.89],[0.000391776,-0.815436,-0.578822,0.00546986],[-1,-1,0,0],[72.8969,9E+09,9E+09,9E+09,9E+09,9E+09]], V_moyen, Z_Xlarge, Tool_defaut;
    MoveJ p_repli, V_moyen, Z_arret, Tool_defaut;
    !
    AutoriseTraj;
    T_Lance;
    !
	ENDPROC

  !-------------------------
  ! Trajectoires de Travail
  !-------------------------

  !-------------
  PROC T_X62E1H1()
    VAR bool bStatus;

    Aff_Traj "T_X62E1H1";
    AntiReboucle;
    !
    !Home Position
    MoveJ p_reb_prg,V_rapide,Z_arret,Tool_defaut\WObj:=wobj0;
    !
    T_SEGURANCATRASEIRA;
    !
    ! E1:autorização de solda 1
    ! O12:fora de interferencia1 com K5
    ! O13:fora de interferencia2 com K5
    EVENT\E1;
    ORDRE\O12\O13;
		!
    AutoriseTraj;
    EVENT\E4;
    T_X62K3E1H1;
    !
    ! O1:fim de solda 1
    ! O12:fora de interferencia1 com K5
    ORDRE\O1\O12;
    !
    ! E2:autorização de solda 2
    ! O12:fora de interferencia1 com K5
    EVENT\E2;
    ORDRE\O12;
    !
    AutoriseTraj;
    T_X62K3E1H1_OP;
    !
    ! O2:fim de solda 2
    ! O12:fora de interferencia1 com K5
    ! O13:fora de interferencia2 com K5
    ORDRE\O2\O12\O13;
    !
    T_AUTORIZA_RECUO;
    !
    !Home Position
    MoveJ p_reb_prg, V_lent, Z_arret, Tool_defaut\WObj:=wobj0;
    !
    T_SEGURANCATRASEIRA;
    !
  ENDPROC

  !-------------
  PROC T_X62E2H2()
    VAR bool bStatus;

    Aff_Traj "T_X62E2H2";
    AntiReboucle;
    !
    !Home Position
    MoveJ p_reb_prg,V_rapide,Z_arret,Tool_defaut\WObj:=wobj0;
    !
    T_SEGURANCATRASEIRA;
    !
    ! E1:autorização de solda 1
    ! O12:fora de interferencia1 com K5
    ! O13:fora de interferencia2 com K5
    EVENT\E1;
    ORDRE\O12\O13;
    !
    AutoriseTraj;
    EVENT\E5;
    T_X62K3E23H2;
    !
    ! O1:fim de solda 1
    ! O12:fora de interferencia1 com K5
    ! O13:fora de interferencia2 com K5
    ORDRE\O1\O12\O13;
    !
    ! E2:autorização de solda 2
    ! O12:fora de interferencia1 com K5
    ! O13:fora de interferencia2 com K5
    EVENT\E2;
    ORDRE\O12\O13;
    !
    AutoriseTraj;
    T_X62K3E23H2_OP;
    !
    ! O2:fim de solda 2
    ! O12:fora de interferencia1 com K5
    ! O13:fora de interferencia2 com K5
    ORDRE\O2\O12\O13;
    !
    T_AUTORIZA_RECUO;
		!
    !Home Position
    MoveJ p_reb_prg,V_rapide,Z_arret,Tool_defaut\WObj:=wobj0;
    !
    T_SEGURANCATRASEIRA;
    !
  ENDPROC

  !-------------
  PROC T_X62E3H2()
    VAR bool bStatus;

    Aff_Traj "T_X62E3H2";
    AntiReboucle;
    !
    !Home Position
    MoveJ p_reb_prg,V_rapide,Z_arret,Tool_defaut\WObj:=wobj0;
    !
    T_SEGURANCATRASEIRA;
    !
    ! E1:autorização de solda 1
    ! O12:fora de interferencia1 com K5
    ! O13:fora de interferencia2 com K5
    EVENT\E1;
    ORDRE\O12\O13;
    !
    AutoriseTraj;
    EVENT\E6;
    T_X62K3E23H2;
    !
    ! O1:fim de solda 1
    ! O12:fora de interferencia1 com K5
    ! O13:fora de interferencia2 com K5
    ORDRE\O1\O12\O13;
    !
    ! E2:autorização de solda 2
    ! O12:fora de interferencia1 com K5
    ! O13:fora de interferencia2 com K5
    ! ABERTURA DOS GRAMPOS
    EVENT\E2;
    ORDRE\O12\O13;
    !
    AutoriseTraj;
    T_X62K3E23H2_OP;
    !
    ! O2:fim de solda 2
    ! O12:fora de interferencia1 com K5
    ! O13:fora de interferencia2 com K5
    ORDRE\O2\O12\O13;
    !
    T_AUTORIZA_RECUO;
    !
    !Home Position
    MoveJ p_reb_prg,V_rapide,Z_arret,Tool_defaut\WObj:=wobj0;
    !
    T_SEGURANCATRASEIRA;
    !
  ENDPROC

  PROC T_X62E3H2B()
    VAR bool bStatus;

    Aff_Traj "T_X62E3H2B";
    AntiReboucle;
    !
    !Home Position
    MoveJ p_reb_prg,V_rapide,Z_arret,Tool_defaut\WObj:=wobj0;
    !
    T_SEGURANCATRASEIRA;
    !
    ! E1:autorização de solda 1
    ! O12:fora de interferencia1 com K5
    ! O13:fora de interferencia2 com K5
    EVENT\E1;
    ORDRE\O12\O13;
    !
    AutoriseTraj;
    EVENT\E7;
    T_X62K3E3H2B;
    !
    ! O1:fim de solda 1
    ! O12:fora de interferencia1 com K5
    ! O13:fora de interferencia2 com K5
    ORDRE\O1\O12\O13;
    !
    ! E2:autorização de solda 2
    ! O12:fora de interferencia1 com K5
    ! O13:fora de interferencia2 com K5
    EVENT\E2;
    ORDRE\O12\O13;
    !
    AutoriseTraj;
    T_X62K3E23H2_OP;
    !
    ! O2:fim de solda 2
    ! O12:fora de interferencia1 com K5
    ! O13:fora de interferencia2 com K5
    ORDRE\O2\O12\O13;
    !
    T_AUTORIZA_RECUO;
    !
    !Home Position
    MoveJ p_reb_prg, V_lent, Z_arret, Tool_defaut\WObj:=wobj0;
    !
    T_SEGURANCATRASEIRA;
    !
  ENDPROC

  !-------------
  PROC T_X62CC()
    VAR bool bStatus;

    Aff_Traj "T_X62CC";
    AntiReboucle;
    !
    !Home Position
    MoveJ p_reb_prg,V_rapide,Z_arret,Tool_defaut\WObj:=wobj0;
    !
    T_SEGURANCATRASEIRA;
    !
    ! E1:autorização de solda 1
    ! O12:fora de interferencia1 com K5
    ! O13:fora de interferencia2 com K5
    EVENT\E1;
    ORDRE\O12\O13;
    !
    AutoriseTraj;
    EVENT\E8;
    T_X62K3CC;
    !
    ! O1:fim de solda 1
    ! O12:fora de interferencia1 com K5
    ! O13:fora de interferencia2 com K5
    ORDRE\O1\O12\O13;
    !
    T_AUTORIZA_RECUO;
    !
    !Home Position
    MoveJ p_reb_prg,V_rapide,Z_arret,Tool_defaut\WObj:=wobj0;
    !
    T_SEGURANCATRASEIRA;
    !
  ENDPROC

  !-------------
  !CASES XDF
  !-------------
    PROC T_XDF_L2H1()
     VAR bool bStatus;

     Aff_Traj "T_XDF_L2H1";
     AntiReboucle;
     !
     !Home Position
     MoveJ p_reb_prg,V_rapide,Z_arret,Tool_defaut\WObj:=wobj0;
     !
     T_SEGURANCATRASEIRA;
     !
     ! E1:autorização de solda 1
     ! O12:fora de interferencia1 com K5
     ! O13:fora de interferencia2 com K5
     ! O14:fora de interferencia3 com K5
     EVENT \E1;
     ORDRE\O12\O13\O14;
     !
     AutoriseTraj;
     EVENT \E8;
     T_SR1_K0_XDF_L2H1;
     !
     ! O1:fim de solda 1
     ! O12:fora de interferencia1 com K5
     ! O13:fora de interferencia2 com K5
     ! O14:fora de interferencia3 com K5
     ORDRE\O1\O12\O13\O14;
     !
     ! E2:autorização de solda 2
     ! O12:fora de interferencia1 com K5
     ! O13:fora de interferencia2 com K5
     ! O14:fora de interferencia3 com K5
     !ABERTURA DE GRAMPOS
     EVENT \E2;
     ORDRE\O12\O13\O14;
     !
     AutoriseTraj;
     EVENT \E8;
     T_SR2_K0_XDF_L2H1;
     !
     ! O2:fim de solda 2
     ! O12:fora de interferencia1 com K5
     ! O13:fora de interferencia2 com K5
     ! O14:fora de interferencia3 com K5
     ORDRE\O2\O12\O13\O14;
     !
     T_AUTORIZA_RECUO;
     !
     !Home Position
     MoveJ p_reb_prg,V_rapide,Z_arret,Tool_defaut\WObj:=wobj0;
     !
     T_SEGURANCATRASEIRA;
     !
  ENDPROC

     !-------------
  PROC T_XDF_L2H2()
     VAR bool bStatus;

     Aff_Traj "T_XDF_L2H1";
     AntiReboucle;
     !
     !Home Position
     MoveJ p_reb_prg,V_rapide,Z_arret,Tool_defaut\Wobj:=wobj0;
     !
     T_SEGURANCATRASEIRA;
     !
     ! E1:autorização de solda 1
     ! O12:fora de interferencia1 com K5
     ! O13:fora de interferencia2 com K5
     ! O14:fora de interferencia3 com K5
     EVENT \E1;
     ORDRE\O12\O13\O14;
     !
     AutoriseTraj;
     EVENT \E5;
     T_SR1_K0_XDF_L2H2;
     !
     ! O1:fim de solda 1
     ! O12:fora de interferencia1 com K5
     ! O13:fora de interferencia2 com K5
     ! O14:fora de interferencia3 com K5
     ORDRE\O1\O12\O13\O14;
     !
     ! E2:autorização de solda 2
     ! O12:fora de interferencia1 com K5
     ! O13:fora de interferencia2 com K5
     ! O14:fora de interferencia3 com K5
     EVENT \E2;
     ORDRE\O12\O13\O14;
     !
     AutoriseTraj;
     T_SR2_K0_XDF_L2H2;
     !
     ! O2:fim de solda 2
     ! O12:fora de interferencia1 com K5
     ! O13:fora de interferencia2 com K5
     ! O14:fora de interferencia3 com K5
     ORDRE\O2\O12\O13\O14;
     !
     ! E3:autorização de solda 3
     ! O12:fora de interferencia1 com K5
     ! O13:fora de interferencia2 com K5
     ! O14:fora de interferencia3 com K5
     EVENT \E3;
     ORDRE\O12\O13\O14;
     !
     AutoriseTraj;
     T_SR3_K0_XDF_L2H2;
     !
     ! O3:fim de solda 3
     ! O12:fora de interferencia1 com K5
     ! O13:fora de interferencia2 com K5
     ! O14:fora de interferencia3 com K5
     ORDRE\O3\O12\O13\O14;
     !
     T_AUTORIZA_RECUO;
     !
     !Home Position
     MoveJ p_reb_prg,V_rapide,Z_arret,Tool_defaut\Wobj:=wobj0;
     !
     T_SEGURANCATRASEIRA;
     !
  ENDPROC

     !-------------
  PROC T_X62K3E1H1()
    VAR bool bStatus;
    Aff_Traj "T_X62K3E1H1";
    AntiReboucle;

    MoveJ pInicioX62_Pinca1, V_rapide, Z_arret, Tool_Pince1\WObj:=wobj_X62;
    !
    ! E13:interferencia2 com K5
    ! O12:fora de interferencia1 com K5
    EVENT\E13;
    ORDRE\O12;
    !
    MoveJ [[602.06,1695.19,2908.36],[0.0694316,-0.00204347,0.00124342,-0.997584],[0,-1,0,0],[59.9379,9E+09,9E+09,9E+09,9E+09,9E+09]], V_rapide, Z_arret, Tool_Pince1\WObj:=wobj_X62;
    !
    ! E13:interferencia2 com K5
    ! O12:fora de interferencia1 com K5
    EVENT\E13;
    ORDRE\O12;
    !
    ! E12:interferencia1 com K5
    EVENT\E12;
    ORDRE;
    !
    MoveJ [[1650.02,1566.66,2799.96],[0.37032,0.00025085,0.00021542,-0.928904],[0,0,1,0],[183.538,9E+09,9E+09,9E+09,9E+09,9E+09]], V_rapide, Z_arret, Tool_Pince1\WObj:=wobj_X62;
    !
    ! E12:interferencia1 com K5
    EVENT\E12;
    ORDRE;
    !
    MoveL [[2334.04,1160.47,2012.84],[0.520616,0.00719435,-0.015037,-0.853628],[0,0,0,0],[86.0789,9E+09,9E+09,9E+09,9E+09,9E+09]], V_rapide, Z_moyen, Tool_Pince1\WObj:=wobj_X62;
    MoveL [[2366.03,960.78,1843.80],[0.579585,0.0017549,-0.0055314,-0.814892],[0,0,0,0],[133.96,9E+09,9E+09,9E+09,9E+09,9E+09]], V_rapide, Z_moyen, Tool_Pince1\WObj:=wobj_X62;
    MoveL [[2275.88,808.64,1827.23],[0.579587,0.00175675,-0.00552378,-0.81489],[0,0,0,0],[153.843,9E+09,9E+09,9E+09,9E+09,9E+09]],V_rapide,Z_Xlarge,Tool_Pince1\WObj:=wobj_X62;
    MoveL [[2296.27,727.79,1826.92],[0.614373,0.000261279,0.000200504,-0.789016],[0,0,0,0],[160,9E+09,9E+09,9E+09,9E+09,9E+09]], V_rapide, Z_Xlarge, Tool_Pince1\WObj:=wobj_X62;
    !
    SR_SOUDER lscs2003267000,V_moyen,1,2,Tool_Pince1,wobj_X62;
    SR_SOUDER lscs2003267100,V_moyen,1,2,Tool_Pince1,wobj_X62;
    SR_SOUDER lscs2003267800,V_moyen,1,2,Tool_Pince1,wobj_X62;
    !
    MoveL [[2458.14,276.89,1941.84],[0.735647,0.000164786,-1.11998E-05,-0.677365],[0,0,0,0],[102.543,9E+09,9E+09,9E+09,9E+09,9E+09]], V_rapide, Z_Xlarge, Tool_Pince1\WObj:=wobj_X62;
    MoveL [[2555.81,169.22,1968.22],[0.842125,-3.9988E-05,2.99759E-05,-0.539283],[0,-1,-1,0],[80.0003,9E+09,9E+09,9E+09,9E+09,9E+09]],V_rapide,Z_Xlarge,Tool_Pince1\WObj:=wobj_X62;
    !
    SR_SOUDER lscs2003267900,V_moyen,1,2,Tool_Pince1,wobj_X62;
    !
    MoveL [[2625.22,701.34,1960.95],[0.924152,-0.00998662,-0.00422478,-0.381871],[0,-1,-1,0],[44.7926,9E+09,9E+09,9E+09,9E+09,9E+09]], V_rapide, Z_Xlarge, Tool_Pince1\WObj:=wobj_X62;
    !
    SR_SOUDER lscs2002842500,V_moyen,1,2,Tool_Pince1,wobj_X62;
    SR_SOUDER lspac002906800,V_moyen,1,1,Tool_Pince1,wobj_X62;
    SR_SOUDER lspac002906700,V_moyen,1,1,Tool_Pince1,wobj_X62;
    SR_SOUDER lspac002906600,V_moyen,1,1,Tool_Pince1,wobj_X62;
    SR_SOUDER lspac006170400,V_moyen,1,1,Tool_Pince1,wobj_X62;
    SR_SOUDER lspac002906400,V_moyen,1,1,Tool_Pince1,wobj_X62;
    SR_SOUDER lspac006171000,V_moyen,1,1,Tool_Pince1,wobj_X62;
    SR_SOUDER lspac002906300,V_moyen,1,1,Tool_Pince1,wobj_X62;
    SR_SOUDER lspac002906200,V_moyen,1,1,Tool_Pince1,wobj_X62;
    SR_SOUDER lspac002906100,V_moyen,1,1,Tool_Pince1,wobj_X62;
    SR_SOUDER lscs1002842300,V_moyen,1,2,Tool_Pince1,wobj_X62;
    !
    MoveL [[2637.11,-638.60,1908.26],[0.781904,0.0244787,0.0194784,-0.622613],[0,0,0,0],[94.9999,9E+09,9E+09,9E+09,9E+09,9E+09]],V_rapide,Z_Xlarge,Tool_Pince1\WObj:=wobj_X62;
    MoveL [[2747.95,-504.11,1917.47],[0.799369,0.0199341,0.0149736,-0.600324],[0,0,0,0],[94.9999,9E+09,9E+09,9E+09,9E+09,9E+09]],V_rapide,Z_Xlarge,Tool_Pince1\WObj:=wobj_X62;
    !
    SR_SOUDER lspac002905100,V_moyen,1,1,Tool_Pince1,wobj_X62;
    SR_SOUDER lscs1002842400,V_moyen,1,2,Tool_Pince1,wobj_X62;
    !
    MoveL [[2790.81,-574.65,1983.86],[0.790295,0.0189822,0.0182127,-0.612162],[0,0,0,0],[40.0003,9E+09,9E+09,9E+09,9E+09,9E+09]],V_rapide,Z_Xlarge,Tool_Pince1\WObj:=wobj_X62;
    MoveL [[2917.59,-580.44,1984.59],[0.797982,4.46834E-05,-2.27802E-05,-0.602681],[0,-1,0,0],[40,9E+09,9E+09,9E+09,9E+09,9E+09]],V_rapide,Z_Xlarge,Tool_Pince1\WObj:=wobj_X62;
    !
    SR_SOUDER lscs1003268200,V_moyen,1,2,Tool_Pince1,wobj_X62;
    SR_SOUDER lscs1003267700,V_moyen,1,2,Tool_Pince1,wobj_X62;
    !
    MoveL [[2860.29,-609.35,1964.91],[0.787351,-2.97805E-07,-5.934E-07,-0.616506],[0,-1,0,0],[35.0002,9E+09,9E+09,9E+09,9E+09,9E+09]],V_rapide,Z_Xlarge,Tool_Pince1\WObj:=wobj_X62;
    MoveL [[2741.48,-625.35,1964.83],[0.787349,2.85529E-05,-2.71971E-05,-0.616508],[0,-1,0,0],[77.1005,9E+09,9E+09,9E+09,9E+09,9E+09]],V_rapide,Z_Xlarge,Tool_Pince1\WObj:=wobj_X62;
    !
    SR_SOUDER lscs1003267600,V_moyen,1,2,Tool_Pince1,wobj_X62;
    !
    MoveL [[2734.18,-712.78,1903.11],[0.787349,3.60883E-05,-2.244E-05,-0.616508],[0,-1,0,0],[114.399,9E+09,9E+09,9E+09,9E+09,9E+09]],V_rapide,Z_Xlarge,Tool_Pince1\WObj:=wobj_X62;
    MoveL [[2616.10,-713.49,1902.92],[0.77085,-3.43978E-07,1.37191E-07,-0.637017],[0,-1,0,0],[118.861,9E+09,9E+09,9E+09,9E+09,9E+09]],V_rapide,Z_Xlarge,Tool_Pince1\WObj:=wobj_X62;
    !
    SR_SOUDER lscs1003267500,V_moyen,1,2,Tool_Pince1,wobj_X62;
    SR_SOUDER lscs1003267400,V_moyen,1,2,Tool_Pince1,wobj_X62;
    SR_SOUDER lscs1003266200,V_moyen,1,2,Tool_Pince1,wobj_X62;
    SR_SOUDER lscs1003266100,V_moyen,1,2,Tool_Pince1,wobj_X62;
    SR_SOUDER lscs1003266000,V_moyen,1,2,Tool_Pince1,wobj_X62;
		!
    ! O12:fora de interferencia1 com K5
    ORDRE\O12;
    !
    SR_SOUDER lscs1002842000,V_moyen,1,2,Tool_Pince1,wobj_X62;
    SR_SOUDER lspac002900900,V_moyen,1,1,Tool_Pince1,wobj_X62;
    SR_SOUDER lspac002901000,V_moyen,1,1,Tool_Pince1,wobj_X62;
    SR_SOUDER lspac002901100,V_moyen,1,1,Tool_Pince1,wobj_X62;
    SR_SOUDER lspac006170500,V_moyen,1,1,Tool_Pince1,wobj_X62;
    SR_SOUDER lspac002901300,V_moyen,1,1,Tool_Pince1,wobj_X62;
    SR_SOUDER lspac006169900,V_moyen,1,1,Tool_Pince1,wobj_X62;
    SR_SOUDER lspac002901600,V_moyen,1,1,Tool_Pince1,wobj_X62;
    SR_SOUDER lspac002901700,V_moyen,1,1,Tool_Pince1,wobj_X62;
    SR_SOUDER lspac002901800,V_moyen,1,1,Tool_Pince1,wobj_X62;
    SR_SOUDER lscs2002842200,V_moyen,1,2,Tool_Pince1,wobj_X62;
    !
    MoveL [[2244.63,704.36,1957.26],[0.614297,-0.0055178,-0.0070443,-0.789024],[0,-1,0,0],[34.9996,9E+09,9E+09,9E+09,9E+09,9E+09]], V_rapide, Z_Xlarge, Tool_Pince1\WObj:=wobj_X62;
    !
    SR_SOUDER lscs2003266900,V_moyen,1,2,Tool_Pince1,wobj_X62;
    !
    MoveL [[2247.79,724.17,1882.37],[0.614379,0.000259899,0.000198438,-0.789011],[0,0,0,0],[110,9E+09,9E+09,9E+09,9E+09,9E+09]],V_rapide,Z_Xlarge,Tool_Pince1\WObj:=wobj_X62;
    MoveL [[2112.32,723.58,1880.50],[0.601153,0.000270135,9.80388E-06,-0.799134],[0,0,0,0],[110,9E+09,9E+09,9E+09,9E+09,9E+09]],V_rapide,Z_Xlarge,Tool_Pince1\WObj:=wobj_X62;
    !
    SR_SOUDER lscs2003266800,V_moyen,1,2,Tool_Pince1,wobj_X62;
    !
    MoveL [[2122.62,678.79,1958.08],[0.601134,-0.0110747,-0.0147027,-0.798936],[0,-1,0,0],[35.0002,9E+09,9E+09,9E+09,9E+09,9E+09]], V_rapide, Z_Xlarge, Tool_Pince1\WObj:=wobj_X62;
    !
    SR_SOUDER lscs2002842100,V_moyen,1,2,Tool_Pince1,wobj_X62;
    SR_SOUDER lspac002904800,V_moyen,1,1,Tool_Pince1,wobj_X62;
    SR_SOUDER lspac002904700,V_moyen,1,1,Tool_Pince1,wobj_X62;
    SR_SOUDER lspac002904600,V_moyen,1,1,Tool_Pince1,wobj_X62;
    SR_SOUDER lspac006170200,V_moyen,1,1,Tool_Pince1,wobj_X62;
    SR_SOUDER lspac002904400,V_moyen,1,1,Tool_Pince1,wobj_X62;
    SR_SOUDER lspac006170800,V_moyen,1,1,Tool_Pince1,wobj_X62;
    SR_SOUDER lspac002904300,V_moyen,1,1,Tool_Pince1,wobj_X62;
    SR_SOUDER lspac002904200,V_moyen,1,1,Tool_Pince1,wobj_X62;
    SR_SOUDER lspac002904100,V_moyen,1,1,Tool_Pince1,wobj_X62;
    SR_SOUDER lscs1002841900,V_moyen,1,2,Tool_Pince1,wobj_X62;
    !
    MoveL [[2120.72,-674.29,1969.84],[0.694652,0.0103914,0.0106962,-0.719191],[0,0,0,0],[34.9999,9E+09,9E+09,9E+09,9E+09,9E+09]], V_rapide, Z_Xlarge, Tool_Pince1\WObj:=wobj_X62;
    !
    SR_SOUDER lscs1003265900,V_moyen,1,2,Tool_Pince1,wobj_X62;
    SR_SOUDER lscs1003265800,V_moyen,1,2,Tool_Pince1,wobj_X62;
    !
    MoveL [[1998.50,-654.29,1964.86],[0.67611,-6.29759E-07,-8.18259E-07,-0.736801],[0,-1,0,0],[40,9E+09,9E+09,9E+09,9E+09,9E+09]],V_rapide,Z_Xlarge,Tool_Pince1\WObj:=wobj_X62;
    MoveL [[1770.89,-653.31,1964.90],[0.641583,9.02895E-05,-4.94446E-05,-0.767053],[0,-1,0,0],[40,9E+09,9E+09,9E+09,9E+09,9E+09]],V_rapide,Z_Xlarge,Tool_Pince1\WObj:=wobj_X62;
    !
    SR_SOUDER lscs1003265600,V_moyen,1,2,Tool_Pince1,wobj_X62;
    SR_SOUDER lscs1003265500,V_moyen,1,2,Tool_Pince1,wobj_X62;
    !
    MoveL [[1682.81,-481.73,1976.88],[0.623823,0.000103804,-6.55606E-05,-0.781566],[0,-1,0,0],[40,9E+09,9E+09,9E+09,9E+09,9E+09]],V_rapide,Z_Xlarge,Tool_Pince1\WObj:=wobj_X62;
    MoveL [[1466.20,-501.73,1976.39],[0.597244,0.000166108,-9.78596E-05,-0.80206],[-1,-1,0,0],[40,9E+09,9E+09,9E+09,9E+09,9E+09]],V_rapide,Z_Xlarge,Tool_Pince1\WObj:=wobj_X62;
    !
    SR_SOUDER lscs1002841500,V_moyen,1,2,Tool_Pince1,wobj_X62;
    SR_SOUDER lspac002878500,V_moyen,1,1,Tool_Pince1,wobj_X62;
    SR_SOUDER lspac002878600,V_moyen,1,1,Tool_Pince1,wobj_X62;
    SR_SOUDER lspac002878700,V_moyen,1,1,Tool_Pince1,wobj_X62;
    SR_SOUDER lspac002878800,V_moyen,1,1,Tool_Pince1,wobj_X62;
    !
    MoveL [[1478.11,-167.48,1999.23],[0.522912,0.00441046,0.00718948,-0.852345],[0,0,0,0],[35,9E+09,9E+09,9E+09,9E+09,9E+09]], V_rapide, Z_Xlarge, Tool_Pince1\WObj:=wobj_X62;
    !
    ! inicio reorientacao
    !
    MoveL [[1480.03,-54.38,1987.71],[0.445099,0.000464,0.001715,-0.89548],[0,0,0,0],[35,35,9E+09,9E+09,9E+09,9E+09]],V_rapide,Z_Xlarge,Tool_Pince1\Wobj:=wobj_X62;
    SR_SOUDER lspac002878900,V_moyen,1,1,Tool_Pince1,wobj_X62;
    SR_SOUDER lspac002879000,V_moyen,1,1,Tool_Pince1,wobj_X62;
    !
    MoveL [[1486,58.82,1993.81],[0.445095,-0.001085,-0.001396,-0.895482],[0,-1,0,0],[35.001,35.001,9E+09,9E+09,9E+09,9E+09]],V_rapide,Z_Xlarge,Tool_Pince1\Wobj:=wobj_X62;
    MoveL [[1486.56,172.72,1985.51],[0.418464,-0.003526,-0.007684,-0.908194],[0,-1,0,0],[35,35,9E+09,9E+09,9E+09,9E+09]],V_rapide,Z_Xlarge,Tool_Pince1\Wobj:=wobj_X62;
    !
    SR_SOUDER lspac002879100,V_moyen,1,1,Tool_Pince1,wobj_X62;
    SR_SOUDER lspac002879200,V_moyen,1,1,Tool_Pince1,wobj_X62;
    SR_SOUDER lspac002879300,V_moyen,1,1,Tool_Pince1,wobj_X62;
    SR_SOUDER lspac002879400,V_moyen,1,1,Tool_Pince1,wobj_X62;
    SR_SOUDER lscs2002841700,V_moyen,1,2,Tool_Pince1,wobj_X62;
    !
    MoveL [[1425.9,638.54,1907.29],[0.294043,-0.009157,-0.029764,-0.955285],[0,-1,0,0],[110,110,9E+09,9E+09,9E+09,9E+09]],V_rapide,Z_Xlarge,Tool_Pince1\Wobj:=wobj_X62;
    MoveL [[1314.4,651.63,1903.47],[0.285707,-0.009481,-0.031761,-0.957744],[0,-1,0,0],[110,110,9E+09,9E+09,9E+09,9E+09]],V_rapide,Z_Xlarge,Tool_Pince1\Wobj:=wobj_X62;
    !
    SR_SOUDER lscs2004621500,V_moyen,1,2,Tool_Pince1,wobj_X62;
    SR_SOUDER lscs2002841600,V_moyen,1,2,Tool_Pince1,wobj_X62;
    SR_SOUDER lspac002883300,V_moyen,1,2,Tool_Pince1,wobj_X62;
    SR_SOUDER lspac002883200,V_moyen,1,2,Tool_Pince1,wobj_X62;
    !
    ! fim reorientacao
    !
    SR_SOUDER lspac002883100,V_moyen,1,2,Tool_Pince1,wobj_X62;
    SR_SOUDER lspac002883000,V_moyen,1,2,Tool_Pince1,wobj_X62;
    !
    MoveL [[1284.37,155.64,1990.63],[0.419394,-0.00275908,-0.00715006,-0.907772],[0,-1,0,0],[34.9999,9E+09,9E+09,9E+09,9E+09,9E+09]],V_rapide,Z_Xlarge,Tool_Pince1\WObj:=wobj_X62;
    !
    SR_SOUDER lspac002882900,V_moyen,1,2,Tool_Pince1,wobj_X62;
    SR_SOUDER lspac002882800,V_moyen,1,2,Tool_Pince1,wobj_X62;
    !
    MoveL [[1278.51,-112.09,1989.48],[0.471233,0.00266987,0.004548,-0.881993],[0,0,0,0],[35.0002,9E+09,9E+09,9E+09,9E+09,9E+09]],V_rapide,Z_Xlarge,Tool_Pince1\WObj:=wobj_X62;
    !
    SR_SOUDER lspac002882700,V_moyen,1,2,Tool_Pince1,wobj_X62;
    SR_SOUDER lspac002882600,V_moyen,1,2,Tool_Pince1,wobj_X62;
    SR_SOUDER lspac002882500,V_moyen,1,2,Tool_Pince1,wobj_X62;
    SR_SOUDER lspac002882400,V_moyen,1,2,Tool_Pince1,wobj_X62;
    SR_SOUDER lscs1002841400, V_moyen, 1, 3, Tool_Pince1, wobj_X62;
    SR_SOUDER lscs1004621400, V_moyen, 1, 3, Tool_Pince1, wobj_X62;
    !
    MoveL [[1326.03,-666.94,1900.90],[0.57702,0.0191693,0.0271029,-0.816055],[-1,0,0,0],[110,9E+09,9E+09,9E+09,9E+09,9E+09]],V_rapide,Z_Xlarge,Tool_Pince1\WObj:=wobj_X62;
    MoveL [[1376.45,-714.23,1896.47],[0.59488,0.0281289,0.0207081,-0.803055],[-1,0,0,0],[110,9E+09,9E+09,9E+09,9E+09,9E+09]],V_rapide,Z_Xlarge,Tool_Pince1\WObj:=wobj_X62;
    !
    SR_SOUDER lscs1005331700,V_moyen,1,2,Tool_Pince1,wobj_X62;
    !
    MoveL [[1377.20,-714.20,1896.45],[0.594883,0.0281337,0.0207115,-0.803053],[-1,0,0,0],[109.998,9E+09,9E+09,9E+09,9E+09,9E+09]],V_rapide,Z_Xlarge,Tool_Pince1\WObj:=wobj_X62;
    MoveL [[1376.88,-653.58,1888.52],[0.583686,0.0278421,0.0211009,-0.811228],[-1,0,0,0],[160,9E+09,9E+09,9E+09,9E+09,9E+09]],V_rapide,Z_Xlarge,Tool_Pince1\WObj:=wobj_X62;
    !
    MoveL [[1472.75,-552.29,1961.43],[0.582477,0.0108645,0.00807295,-0.812735],[0,0,0,0],[173.549,9E+09,9E+09,9E+09,9E+09,9E+09]],V_rapide,Z_Xlarge,Tool_Pince1\WObj:=wobj_X62;
    MoveL [[1677.02,66.13,1941.27],[0.512932,0.000248194,-7.61386E-05,-0.858429],[0,0,0,0],[90.0001,9E+09,9E+09,9E+09,9E+09,9E+09]],V_rapide,Z_Xlarge,Tool_Pince1\WObj:=wobj_X62;
    !
    SR_SOUDER lscsd004573702,V_moyen,1,2,Tool_Pince1,wobj_X62;
    SR_SOUDER lscs2003266400,V_moyen,1,2,Tool_Pince1,wobj_X62;
    SR_SOUDER lscs2003266500,V_moyen,1,2,Tool_Pince1,wobj_X62;
    !
    MoveL [[1770.63,633.16,1964.83],[0.41249,0.000311019,0.000100084,-0.910962],[0,0,0,0],[39.9093,9E+09,9E+09,9E+09,9E+09,9E+09]],V_rapide,Z_Xlarge,Tool_Pince1\WObj:=wobj_X62;
    MoveL [[1998.59,635.60,1964.31],[0.518079,0.000314988,5.76045E-05,-0.855333],[0,0,0,0],[39.9997,9E+09,9E+09,9E+09,9E+09,9E+09]],V_rapide,Z_Xlarge,Tool_Pince1\WObj:=wobj_X62;
    !
    SR_SOUDER lscs2003266700,V_moyen,1,2,Tool_Pince1,wobj_X62;
    ! Abrir grampos
    !
  ENDPROC

  !-------------
  PROC T_X62K3E1H1_OP()
    VAR bool bStatus;
    Aff_Traj "T_X62K3E1H1_OP";
    AntiReboucle;
    !
    MoveL [[1884.13,727.83,1956.34],[0.460207,3.13892E-07,2.91406E-06,-0.887812],[0,0,0,0],[74.9997,9E+09,9E+09,9E+09,9E+09,9E+09]], V_rapide, Z_arret, Tool_Pince1\WObj:=wobj_X62;
    !
    SR_SOUDER lscs2003266600,V_moyen,1,2,Tool_Pince1,wobj_X62;
    !
    MoveL [[1884.65,-13.29,1966.91],[0.640557,0.000108551,-5.50037E-05,-0.767911],[0,-1,0,0],[80.0001,9E+09,9E+09,9E+09,9E+09,9E+09]],V_rapide,Z_Xlarge,Tool_Pince1\WObj:=wobj_X62;
    MoveL [[2185.91,-250.98,1919.46],[0.692856,0.00161498,-0.00123207,-0.721073],[0,0,0,0],[100.206,9E+09,9E+09,9E+09,9E+09,9E+09]], V_rapide, Z_Xlarge, Tool_Pince1\WObj:=wobj_X62;
    MoveL [[2683.28,-643.30,1891.35],[0.771625,0.00407075,-0.00318061,-0.636057],[0,0,0,0],[133.574,9E+09,9E+09,9E+09,9E+09,9E+09]], V_rapide, Z_Xlarge, Tool_Pince1\WObj:=wobj_X62;
    MoveL [[2779.01,-718.78,1902.38],[0.785632,0.00453993,-0.00354845,-0.618667],[0,0,0,0],[140,9E+09,9E+09,9E+09,9E+09,9E+09]], V_rapide, Z_Xlarge, Tool_Pince1\WObj:=wobj_X62;
    !
    SR_SOUDER lscs2003266600_1, V_moyen, 1, 2, Tool_Pince1, wobj_X62;
    !
    MoveL [[2779.01,-718.78,1902.38],[0.785632,0.00453979,-0.00354866,-0.618667],[0,0,0,0],[140,9E+09,9E+09,9E+09,9E+09,9E+09]], V_rapide, Z_Xlarge, Tool_Pince1\WObj:=wobj_X62;
    MoveL [[2683.28,-643.30,1891.35],[0.771625,0.00407075,-0.00318061,-0.636057],[0,0,0,0],[133.574,9E+09,9E+09,9E+09,9E+09,9E+09]], V_rapide, Z_Xlarge, Tool_Pince1\WObj:=wobj_X62;
    MoveL [[2683.28,-643.30,1891.35],[0.771625,0.00407075,-0.00318061,-0.636057],[0,0,0,0],[133.574,9E+09,9E+09,9E+09,9E+09,9E+09]], V_rapide, Z_Xlarge, Tool_Pince1\WObj:=wobj_X62;
    MoveL [[1884.65,-13.29,1966.91],[0.640557,0.000108551,-5.50037E-05,-0.767911],[0,-1,0,0],[80.0001,9E+09,9E+09,9E+09,9E+09,9E+09]],V_rapide,Z_Xlarge,Tool_Pince1\WObj:=wobj_X62;
    !
    SR_SOUDER lscs1003265700,V_moyen,1,2,Tool_Pince1,wobj_X62;
    !
    MoveL [[1514.88,-643.06,1947.44],[0.5925,9.27189E-05,-6.68039E-05,-0.805571],[0,-1,0,0],[149.3,9E+09,9E+09,9E+09,9E+09,9E+09]],V_rapide,Z_Xlarge,Tool_Pince1\WObj:=wobj_X62;
    !
    SR_SOUDER lscsg004573701,V_moyen,1,2,Tool_Pince1,wobj_X62;
    !
    MoveL [[1884.65,-13.30,1954.76],[0.618166,0.000104828,-6.18333E-05,-0.786048],[0,-1,0,0],[80.0006,9E+09,9E+09,9E+09,9E+09,9E+09]],V_rapide,Z_Xlarge,Tool_Pince1\WObj:=wobj_X62;
    MoveL [[1998.64,723.67,1861.81],[0.512721,0.00031549,6.58932E-05,-0.858555],[0,0,0,0],[160,9E+09,9E+09,9E+09,9E+09,9E+09]],V_rapide,Z_Xlarge,Tool_Pince1\WObj:=wobj_X62;
    MoveL [[1969.28,793.00,1829.07],[0.489469,0.000305124,0.000104824,-0.872021],[0,0,0,0],[160,9E+09,9E+09,9E+09,9E+09,9E+09]],V_rapide,Z_Xlarge,Tool_Pince1\WObj:=wobj_X62;
    MoveL [[2110.74,1024.86,1824.65],[0.489468,0.000306777,9.98249E-05,-0.872021],[0,0,0,0],[160,9E+09,9E+09,9E+09,9E+09,9E+09]], V_rapide, Z_moyen, Tool_Pince1\WObj:=wobj_X62;
    MoveL [[2056.27,946.78,3151.45],[0.489467,0.000307522,9.8687E-05,-0.872022],[0,0,0,0],[160,9E+09,9E+09,9E+09,9E+09,9E+09]], V_moyen, Z_Xlarge, Tool_Pince1\WObj:=wobj_X62;
    MoveJ [[1313.96,1370.91,3121.55],[0.18712,0.000204623,-0.00167684,-0.982336],[0,0,1,0],[128.401,9E+09,9E+09,9E+09,9E+09,9E+09]], V_moyen, Z_arret, Tool_Pince1\WObj:=wobj_X62;
    MoveJ pInicioX62_Pinca1, V_moyen, Z_arret, Tool_Pince1\WObj:=wobj_X62;
    !
  ENDPROC

  !-------------
  PROC T_X62K3E3H2B()
    VAR bool bStatus;
    Aff_Traj "T_X62K3E3H2B";
    AntiReboucle;

